SPLINE
SPL {X  -165.650, Y  +471.956, Z    +0.000, E1   -39.047, E3 +385632.686}
SPL {X  -165.650, Y  +478.019, Z    +0.000, E1   -39.139, E3 +385647.571}
SPL {X  -165.650, Y  +484.115, Z    +0.000, E1   -39.050, E3 +385663.332}
SPL {X  -165.650, Y  +488.489, Z    +0.000, E1   -39.102, E3 +385673.940}
SPL {X  -165.650, Y  +491.785, Z    +0.000, E1   -39.157, E3 +385681.913}
SPL {X  -165.650, Y  +496.519, Z    +0.000, E1   -39.062, E3 +385694.527}
SPL {X  -165.650, Y  +501.480, Z    +0.000, E1   -39.099, E3 +385706.684}
SPL {X  -165.650, Y  +505.989, Z    +0.000, E1   -39.067, E3 +385718.316}
SPL {X  -165.650, Y  +512.188, Z    +0.000, E1   -39.077, E3 +385733.959}
SPL {X  -165.650, Y  +516.634, Z    +0.000, E1   -39.035, E3 +385745.205}
SPL {X  -165.650, Y  +521.541, Z    +0.000, E1   -39.052, E3 +385757.752}
SPL {X  -165.650, Y  +527.474, Z    +0.000, E1   -39.169, E3 +385771.770}
SPL {X  -165.650, Y  +532.836, Z    +0.000, E1   -39.150, E3 +385785.552}
SPL {X  -165.650, Y  +537.667, Z    +0.000, E1   -38.986, E3 +385798.497}
SPL {X  -165.650, Y  +542.804, Z    +0.000, E1   -39.141, E3 +385810.681}
SPL {X  -165.650, Y  +547.280, Z    +0.000, E1   -38.965, E3 +385822.826}
SPL {X  -165.650, Y  +551.666, Z    +0.000, E1   -39.102, E3 +385833.144}
SPL {X  -165.650, Y  +557.612, Z    +0.000, E1   -39.166, E3 +385847.790}
SPL {X  -165.650, Y  +562.850, Z    +0.000, E1   -38.959, E3 +385862.149}
SPL {X  -165.650, Y  +568.257, Z    +0.000, E1   -39.077, E3 +385875.104}
SPL {X  -165.650, Y  +573.200, Z    +0.000, E1   -39.061, E3 +385887.639}
SPL {X  -165.650, Y  +578.240, Z    +0.000, E1   -39.117, E3 +385899.980}
SPL {X  -165.650, Y  +582.804, Z    +0.000, E1   -39.080, E3 +385911.687}
SPL {X  -165.650, Y  +587.640, Z    +0.000, E1   -39.069, E3 +385923.944}
SPL {X  -165.650, Y  +593.610, Z    +0.000, E1   -39.204, E3 +385938.217}
SPL {X  -165.650, Y  +599.021, Z    +0.000, E1   -38.950, E3 +385953.367}
SPL {X  -165.650, Y  +604.635, Z    +0.000, E1   -39.163, E3 +385966.144}
SPL {X  -165.650, Y  +608.365, Z    +0.000, E1   -39.063, E3 +385976.134}
SPL {X  -165.650, Y  +612.142, Z    +0.000, E1   -39.023, E3 +385985.864}
SPL {X  -165.650, Y  +616.635, Z    +0.000, E1   -39.260, E3 +385995.751}
SPL {X  -165.650, Y  +620.299, Z    +0.000, E1   -38.904, E3 +386007.138}
SPL {X  -165.650, Y  +625.662, Z    +0.000, E1   -39.189, E3 +386018.949}
SPL {X  -165.650, Y  +629.982, Z    +0.000, E1   -39.063, E3 +386030.550}
SPL {X  -165.650, Y  +635.019, Z    +0.000, E1   -39.106, E3 +386043.032}
SPL {X  -165.650, Y  +641.706, Z    +0.000, E1   -39.097, E3 +386060.099}
SPL {X  -165.650, Y  +648.294, Z    +0.000, E1   -39.142, E3 +386076.222}
SPL {X  -165.650, Y  +652.477, Z    +0.000, E1   -39.068, E3 +386087.124}
SPL {X  -165.650, Y  +656.920, Z    +0.000, E1   -39.120, E3 +386098.079}
SPL {X  -165.650, Y  +661.125, Z    +0.000, E1   -39.092, E3 +386108.728}
SPL {X  -165.650, Y  +664.437, Z    +0.000, E1   -39.114, E3 +386116.937}
SPL {X  -165.650, Y  +668.296, Z    +0.000, E1   -39.077, E3 +386126.909}
SPL {X  -165.650, Y  +673.138, Z    +0.000, E1   -39.196, E3 +386138.365}
SPL {X  -165.640, Y  +677.281, Z    +0.000, E1   -38.803, E3 +386151.254}
SPL {X  -165.389, Y  +684.794, Z    +0.000, E1   -39.261, E3 +386167.564}
SPL {X  -164.948, Y  +690.736, Z    +0.000, E1   -38.951, E3 +386184.233}
SPL {X  -164.363, Y  +696.109, Z    +0.000, E1   -38.853, E3 +386198.324}
SPL {X  -163.795, Y  +700.218, Z    +0.000, E1   -38.698, E3 +386209.531}
SPL {X  -162.937, Y  +705.358, Z    +0.000, E1   -38.703, E3 +386222.599}
SPL {X  -161.983, Y  +710.160, Z    +0.000, E1   -38.439, E3 +386236.093}
SPL {X  -161.163, Y  +713.794, Z    +0.000, E1   -38.390, E3 +386245.463}
SPL {X  -160.158, Y  +717.801, Z    +0.000, E1   -38.225, E3 +386256.593}
SPL {X  -155.870, Y  +731.575, Z    +0.000, E1   -42.661, E3 +386264.056}
SPL {X  -137.799, Y  +767.431, Z    +0.000, E1   -46.550, E3 +386320.566}
ENDSPLINE

SPLINE
SPL {X  -141.948, Y  +760.885, Z    +0.000, E1   -42.258, E3 +386352.702}
SPL {X  -160.264, Y  +717.397, Z    +0.000, E1   -24.835, E3 +386393.887}
SPL {X  -164.762, Y  +692.628, Z    +0.000, E1   -12.660, E3 +386397.139}
SPL {X  -165.581, Y  +680.274, Z    +0.000, E1    -5.699, E3 +386392.624}
SPL {X  -165.650, Y  +673.662, Z    +0.000, E1    -1.458, E3 +386389.583}
SPL {X  -165.650, Y  +670.254, Z    +0.000, E1    +1.045, E3 +386391.947}
SPL {X  -165.650, Y  +666.842, Z    +0.000, E1    +3.871, E3 +386390.049}
SPL {X  -165.650, Y  +661.513, Z    +0.000, E1    +8.695, E3 +386389.957}
SPL {X  -165.650, Y  +654.973, Z    +0.000, E1   +15.752, E3 +386387.363}
SPL {X  -165.650, Y  +648.120, Z    +0.000, E1   +22.794, E3 +386387.475}
SPL {X  -165.650, Y  +632.103, Z    +0.000, E1   +42.949, E3 +386374.433}
SPL {X  -165.650, Y  +609.948, Z    +0.000, E1   +49.636, E3 +386391.859}
SPL {X  -165.650, Y  +601.895, Z    +0.000, E1   +47.595, E3 +386409.529}
SPL {X  -165.650, Y  +568.828, Z    +0.000, E1   +48.639, E3 +386457.284}
ENDSPLINE

SPLINE
SPL {X  -165.650, Y  +587.144, Z    +0.000, E1   +39.840, E3 +386471.316}
ENDSPLINE

SPLINE
SPL {X  -165.650, Y  +582.480, Z    +0.000, E1   +38.929, E3 +386488.512}
SPL {X  -165.650, Y  +575.679, Z    +0.000, E1   +38.947, E3 +386505.587}
SPL {X  -165.650, Y  +569.616, Z    +0.000, E1   +38.966, E3 +386520.746}
SPL {X  -165.650, Y  +564.364, Z    +0.000, E1   +38.909, E3 +386534.398}
SPL {X  -165.650, Y  +559.065, Z    +0.000, E1   +38.883, E3 +386547.976}
SPL {X  -165.650, Y  +552.770, Z    +0.000, E1   +38.963, E3 +386563.537}
SPL {X  -165.650, Y  +546.277, Z    +0.000, E1   +38.910, E3 +386580.279}
SPL {X  -165.650, Y  +540.151, Z    +0.000, E1   +38.996, E3 +386595.208}
SPL {X  -165.650, Y  +534.008, Z    +0.000, E1   +38.962, E3 +386611.050}
SPL {X  -165.650, Y  +528.320, Z    +0.000, E1   +38.809, E3 +386626.287}
SPL {X  -165.650, Y  +522.377, Z    +0.000, E1   +38.974, E3 +386640.406}
ENDSPLINE

SPLINE
SPL {X  -165.650, Y  +539.854, Z    +0.000, E1   +28.090, E3 +386657.023}
ENDSPLINE

SPLINE
SPL {X  -165.650, Y  +534.443, Z    +0.000, E1   +28.969, E3 +386671.075}
SPL {X  -165.650, Y  +530.452, Z    +0.000, E1   +29.664, E3 +386680.808}
SPL {X  -165.650, Y  +525.298, Z    +0.000, E1   +30.602, E3 +386692.618}
SPL {X  -165.650, Y  +518.290, Z    +0.000, E1   +31.783, E3 +386708.511}
SPL {X  -165.650, Y  +512.706, Z    +0.000, E1   +32.573, E3 +386721.345}
SPL {X  -165.650, Y  +507.785, Z    +0.000, E1   +33.438, E3 +386731.282}
SPL {X  -165.650, Y  +501.257, Z    +0.000, E1   +34.478, E3 +386744.522}
SPL {X  -165.650, Y  +493.800, Z    +0.000, E1   +35.486, E3 +386760.010}
SPL {X  -165.650, Y  +485.583, Z    +0.000, E1   +36.670, E3 +386775.733}
SPL {X  -165.650, Y  +477.375, Z    +0.000, E1   +37.747, E3 +386791.252}
SPL {X  -165.650, Y  +469.901, Z    +0.000, E1   +38.767, E3 +386804.384}
SPL {X  -165.650, Y  +463.507, Z    +0.000, E1   +39.800, E3 +386814.131}
SPL {X  -165.650, Y  +460.803, Z    +0.000, E1   +39.417, E3 +386823.195}
SPL {X  -165.650, Y  +455.681, Z    +0.000, E1   +39.641, E3 +386834.516}
SPL {X  -165.650, Y  +451.332, Z    +0.000, E1   +39.738, E3 +386844.648}
SPL {X  -165.650, Y  +448.050, Z    +0.000, E1   +39.392, E3 +386854.814}
SPL {X  -165.650, Y  +442.946, Z    +0.000, E1   +39.866, E3 +386864.589}
SPL {X  -165.650, Y  +439.091, Z    +0.000, E1   +39.674, E3 +386875.207}
SPL {X  -165.650, Y  +434.131, Z    +0.000, E1   +39.643, E3 +386887.719}
SPL {X  -165.650, Y  +428.810, Z    +0.000, E1   +39.691, E3 +386900.482}
SPL {X  -165.650, Y  +424.197, Z    +0.000, E1   +39.695, E3 +386911.840}
SPL {X  -165.650, Y  +420.220, Z    +0.000, E1   +39.526, E3 +386922.635}
SPL {X  -165.650, Y  +414.177, Z    +0.000, E1   +39.693, E3 +386936.762}
SPL {X  -165.650, Y  +407.394, Z    +0.000, E1   +39.797, E3 +386952.717}
SPL {X  -165.650, Y  +402.798, Z    +0.000, E1   +39.651, E3 +386964.838}
SPL {X  -165.650, Y  +398.253, Z    +0.000, E1   +39.688, E3 +386975.842}
SPL {X  -165.650, Y  +393.720, Z    +0.000, E1   +39.686, E3 +386987.016}
SPL {X  -165.650, Y  +389.210, Z    +0.000, E1   +39.696, E3 +386998.066}
SPL {X  -165.650, Y  +384.878, Z    +0.000, E1   +39.631, E3 +387009.142}
SPL {X  -165.650, Y  +380.529, Z    +0.000, E1   +39.528, E3 +387020.529}
SPL {X  -165.618, Y  +375.240, Z    +0.000, E1   +39.617, E3 +387033.123}
SPL {X  -165.428, Y  +369.922, Z    +0.000, E1   +39.705, E3 +387045.664}
SPL {X  -165.216, Y  +366.519, Z    +0.000, E1   +39.498, E3 +387055.231}
SPL {X  -164.790, Y  +361.646, Z    +0.000, E1   +39.684, E3 +387066.226}
SPL {X  -164.317, Y  +357.530, Z    +0.000, E1   +39.402, E3 +387077.939}
SPL {X  -163.775, Y  +353.645, Z    +0.000, E1   +39.313, E3 +387088.110}
SPL {X  -163.109, Y  +349.595, Z    +0.000, E1   +39.290, E3 +387098.172}
SPL {X  -162.309, Y  +345.398, Z    +0.000, E1   +39.085, E3 +387109.835}
SPL {X  -161.467, Y  +341.510, Z    +0.000, E1   +38.980, E3 +387119.881}
SPL {X  -160.812, Y  +338.758, Z    +0.000, E1   +38.898, E3 +387127.138}
SPL {X  -159.926, Y  +335.332, Z    +0.000, E1   +38.809, E3 +387136.095}
SPL {X  -153.020, Y  +315.059, Z    +0.000, E1   +45.580, E3 +387142.827}
SPL {X  -148.632, Y  +305.368, Z    +0.000, E1   +40.700, E3 +387202.428}
SPL {X  -145.004, Y  +298.414, Z    +0.000, E1   +40.971, E3 +387227.164}
ENDSPLINE

SPLINE
SPL {X  -149.687, Y  +307.551, Z    +0.000, E1   +36.303, E3 +387262.596}
SPL {X  -158.807, Y  +331.381, Z    +0.000, E1   +26.928, E3 +387286.249}
SPL {X  -164.505, Y  +359.058, Z    +0.000, E1   +13.887, E3 +387275.010}
SPL {X  -165.494, Y  +371.321, Z    +0.000, E1    +7.176, E3 +387273.571}
SPL {X  -165.650, Y  +379.419, Z    +0.000, E1    +2.065, E3 +387271.252}
SPL {X  -165.650, Y  +383.176, Z    +0.000, E1    -0.610, E3 +387272.247}
SPL {X  -165.650, Y  +388.696, Z    +0.000, E1    -5.134, E3 +387270.524}
SPL {X  -165.650, Y  +394.663, Z    +0.000, E1   -10.843, E3 +387271.680}
SPL {X  -165.650, Y  +400.450, Z    +0.000, E1   -18.287, E3 +387262.979}
SPL {X  -165.650, Y  +409.248, Z    +0.000, E1   -26.478, E3 +387266.602}
SPL {X  -165.650, Y  +418.660, Z    +0.000, E1   -36.186, E3 +387264.078}
SPL {X  -165.650, Y  +444.260, Z    +0.000, E1   -47.328, E3 +387279.826}
SPL {X  -165.650, Y  +458.981, Z    +0.000, E1   -49.189, E3 +387295.369}
SPL {X  -165.650, Y  +493.049, Z    +0.000, E1   -51.657, E3 +387334.402}
ENDSPLINE

SPLINE
SPL {X  -165.650, Y  +468.984, Z    +0.000, E1   -41.461, E3 +387347.262}
SPL {X  -165.650, Y  +467.052, Z    +0.000, E1   -38.928, E3 +387357.877}
ENDSPLINE

SPLINE
SPL {X  -165.650, Y  +471.956, Z    +0.000, E1   -39.047, E3 +387369.528}
SPL {X  -165.650, Y  +478.019, Z    +0.000, E1   -39.139, E3 +387384.413}
SPL {X  -165.650, Y  +484.115, Z    +0.000, E1   -39.050, E3 +387400.174}
SPL {X  -165.650, Y  +490.374, Z    +0.000, E1   -39.169, E3 +387415.294}
SPL {X  -165.650, Y  +495.141, Z    +0.000, E1   -39.109, E3 +387427.450}
SPL {X  -165.650, Y  +497.824, Z    +0.000, E1   -38.944, E3 +387435.208}
SPL {X  -165.650, Y  +502.351, Z    +0.000, E1   -39.056, E3 +387446.092}
SPL {X  -165.650, Y  +508.180, Z    +0.000, E1   -39.157, E3 +387460.158}
SPL {X  -165.650, Y  +513.074, Z    +0.000, E1   -38.997, E3 +387473.375}
SPL {X  -165.650, Y  +518.439, Z    +0.000, E1   -39.071, E3 +387486.526}
SPL {X  -165.650, Y  +523.032, Z    +0.000, E1   -38.966, E3 +387498.662}
SPL {X  -165.650, Y  +528.401, Z    +0.000, E1   -39.135, E3 +387511.262}
SPL {X  -165.650, Y  +533.857, Z    +0.000, E1   -39.163, E3 +387524.768}
SPL {X  -165.650, Y  +539.651, Z    +0.000, E1   -39.087, E3 +387539.912}
SPL {X  -165.650, Y  +544.603, Z    +0.000, E1   -39.103, E3 +387552.088}
SPL {X  -165.650, Y  +547.280, Z    +0.000, E1   -38.965, E3 +387559.668}
SPL {X  -165.650, Y  +551.666, Z    +0.000, E1   -39.102, E3 +387569.986}
SPL {X  -165.650, Y  +555.880, Z    +0.000, E1   -39.094, E3 +387580.557}
SPL {X  -165.650, Y  +559.255, Z    +0.000, E1   -39.167, E3 +387588.593}
SPL {X  -165.650, Y  +562.850, Z    +0.000, E1   -38.959, E3 +387598.991}
SPL {X  -165.650, Y  +568.257, Z    +0.000, E1   -39.077, E3 +387611.946}
SPL {X  -165.650, Y  +573.200, Z    +0.000, E1   -39.061, E3 +387624.481}
SPL {X  -165.650, Y  +578.240, Z    +0.000, E1   -39.117, E3 +387636.822}
SPL {X  -165.650, Y  +582.804, Z    +0.000, E1   -39.080, E3 +387648.529}
SPL {X  -165.650, Y  +587.640, Z    +0.000, E1   -39.069, E3 +387660.786}
SPL {X  -165.650, Y  +593.610, Z    +0.000, E1   -39.204, E3 +387675.060}
SPL {X  -165.650, Y  +599.021, Z    +0.000, E1   -38.950, E3 +387690.209}
SPL {X  -165.650, Y  +604.635, Z    +0.000, E1   -39.163, E3 +387702.986}
SPL {X  -165.650, Y  +608.365, Z    +0.000, E1   -39.063, E3 +387712.976}
SPL {X  -165.650, Y  +612.142, Z    +0.000, E1   -39.023, E3 +387722.706}
SPL {X  -165.650, Y  +616.635, Z    +0.000, E1   -39.260, E3 +387732.593}
SPL {X  -165.650, Y  +620.299, Z    +0.000, E1   -38.904, E3 +387743.980}
SPL {X  -165.650, Y  +625.662, Z    +0.000, E1   -39.189, E3 +387755.791}
SPL {X  -165.650, Y  +629.982, Z    +0.000, E1   -39.063, E3 +387767.392}
SPL {X  -165.650, Y  +635.019, Z    +0.000, E1   -39.106, E3 +387779.874}
SPL {X  -165.650, Y  +640.403, Z    +0.000, E1   -39.127, E3 +387793.270}
SPL {X  -165.650, Y  +645.443, Z    +0.000, E1   -39.032, E3 +387806.575}
SPL {X  -165.650, Y  +651.452, Z    +0.000, E1   -39.128, E3 +387821.144}
SPL {X  -165.650, Y  +656.920, Z    +0.000, E1   -39.120, E3 +387834.921}
SPL {X  -165.650, Y  +661.125, Z    +0.000, E1   -39.092, E3 +387845.570}
SPL {X  -165.650, Y  +664.437, Z    +0.000, E1   -39.114, E3 +387853.779}
SPL {X  -165.650, Y  +668.296, Z    +0.000, E1   -39.077, E3 +387863.751}
SPL {X  -165.650, Y  +673.138, Z    +0.000, E1   -39.196, E3 +387875.207}
SPL {X  -165.640, Y  +677.281, Z    +0.000, E1   -38.803, E3 +387888.096}
SPL {X  -165.461, Y  +683.414, Z    +0.000, E1   -39.212, E3 +387901.080}
SPL {X  -165.241, Y  +687.126, Z    +0.000, E1   -39.221, E3 +387910.223}
SPL {X  -164.948, Y  +690.736, Z    +0.000, E1   -38.951, E3 +387921.075}
SPL {X  -164.363, Y  +696.109, Z    +0.000, E1   -38.853, E3 +387935.166}
SPL {X  -163.795, Y  +700.218, Z    +0.000, E1   -38.698, E3 +387946.373}
SPL {X  -162.937, Y  +705.358, Z    +0.000, E1   -38.703, E3 +387959.441}
SPL {X  -161.983, Y  +710.160, Z    +0.000, E1   -38.439, E3 +387972.935}
SPL {X  -160.874, Y  +714.989, Z    +0.000, E1   -38.205, E3 +387986.596}
SPL {X  -159.557, Y  +720.012, Z    +0.000, E1   -38.534, E3 +387997.137}
SPL {X  -155.870, Y  +731.575, Z    +0.000, E1   -42.661, E3 +388000.898}
SPL {X  -137.799, Y  +767.431, Z    +0.000, E1   -46.550, E3 +388057.408}
ENDSPLINE

SPLINE
SPL {X  -141.948, Y  +760.885, Z    +0.000, E1   -42.258, E3 +388089.544}
SPL {X  -160.264, Y  +717.397, Z    +0.000, E1   -24.835, E3 +388130.729}
SPL {X  -164.457, Y  +695.345, Z    +0.000, E1   -14.031, E3 +388137.670}
SPL {X  -165.312, Y  +686.072, Z    +0.000, E1    -9.096, E3 +388130.764}
SPL {X  -165.625, Y  +678.398, Z    +0.000, E1    -4.508, E3 +388128.506}
SPL {X  -165.650, Y  +673.662, Z    +0.000, E1    -1.458, E3 +388126.425}
SPL {X  -165.650, Y  +670.254, Z    +0.000, E1    +1.045, E3 +388128.789}
SPL {X  -165.650, Y  +666.842, Z    +0.000, E1    +3.871, E3 +388126.891}
SPL {X  -165.650, Y  +662.773, Z    +0.000, E1    +7.549, E3 +388127.036}
SPL {X  -165.650, Y  +656.581, Z    +0.000, E1   +13.870, E3 +388125.086}
SPL {X  -165.650, Y  +648.120, Z    +0.000, E1   +22.794, E3 +388124.317}
SPL {X  -165.650, Y  +632.103, Z    +0.000, E1   +42.949, E3 +388111.275}
SPL {X  -165.650, Y  +609.948, Z    +0.000, E1   +49.636, E3 +388128.701}
SPL {X  -165.650, Y  +601.895, Z    +0.000, E1   +47.595, E3 +388146.371}
SPL {X  -165.650, Y  +568.828, Z    +0.000, E1   +48.639, E3 +388194.126}
ENDSPLINE

SPLINE
SPL {X  -165.650, Y  +587.144, Z    +0.000, E1   +39.840, E3 +388208.158}
ENDSPLINE

SPLINE
SPL {X  -165.650, Y  +582.480, Z    +0.000, E1   +38.929, E3 +388225.354}
SPL {X  -165.650, Y  +576.923, Z    +0.000, E1   +38.908, E3 +388239.384}
SPL {X  -165.650, Y  +570.800, Z    +0.000, E1   +39.001, E3 +388254.559}
SPL {X  -165.650, Y  +564.364, Z    +0.000, E1   +38.909, E3 +388271.241}
SPL {X  -165.650, Y  +559.065, Z    +0.000, E1   +38.883, E3 +388284.819}
SPL {X  -165.650, Y  +554.358, Z    +0.000, E1   +38.887, E3 +388296.660}
SPL {X  -165.650, Y  +549.409, Z    +0.000, E1   +38.884, E3 +388309.341}
SPL {X  -165.650, Y  +542.772, Z    +0.000, E1   +39.054, E3 +388325.137}
SPL {X  -165.650, Y  +537.647, Z    +0.000, E1   +38.838, E3 +388339.299}
SPL {X  -165.650, Y  +532.636, Z    +0.000, E1   +39.009, E3 +388350.945}
SPL {X  -165.650, Y  +528.320, Z    +0.000, E1   +38.809, E3 +388363.129}
SPL {X  -165.650, Y  +522.377, Z    +0.000, E1   +38.974, E3 +388377.249}
ENDSPLINE

SPLINE
SPL {X  -165.650, Y  +541.168, Z    +0.000, E1   +27.957, E3 +388389.588}
ENDSPLINE

SPLINE
SPL {X  -165.650, Y  +536.052, Z    +0.000, E1   +28.653, E3 +388404.223}
SPL {X  -165.650, Y  +530.452, Z    +0.000, E1   +29.664, E3 +388417.650}
SPL {X  -165.650, Y  +523.712, Z    +0.000, E1   +30.911, E3 +388432.932}
SPL {X  -165.650, Y  +516.975, Z    +0.000, E1   +31.942, E3 +388448.526}
SPL {X  -165.650, Y  +512.706, Z    +0.000, E1   +32.573, E3 +388458.187}
SPL {X  -165.650, Y  +507.785, Z    +0.000, E1   +33.438, E3 +388468.124}
SPL {X  -165.650, Y  +501.257, Z    +0.000, E1   +34.478, E3 +388481.364}
SPL {X  -165.650, Y  +495.236, Z    +0.000, E1   +35.288, E3 +388493.870}
SPL {X  -165.650, Y  +488.684, Z    +0.000, E1   +36.217, E3 +388506.766}
SPL {X  -165.650, Y  +481.130, Z    +0.000, E1   +37.251, E3 +388521.075}
SPL {X  -165.650, Y  +475.455, Z    +0.000, E1   +37.964, E3 +388531.732}
SPL {X  -165.650, Y  +469.901, Z    +0.000, E1   +38.767, E3 +388541.226}
SPL {X  -165.650, Y  +465.276, Z    +0.000, E1   +39.067, E3 +388551.103}
SPL {X  -165.650, Y  +459.623, Z    +0.000, E1   +39.919, E3 +388560.038}
SPL {X  -165.650, Y  +455.681, Z    +0.000, E1   +39.641, E3 +388571.358}
SPL {X  -165.650, Y  +451.332, Z    +0.000, E1   +39.738, E3 +388581.491}
SPL {X  -165.650, Y  +448.050, Z    +0.000, E1   +39.392, E3 +388591.656}
SPL {X  -165.650, Y  +442.946, Z    +0.000, E1   +39.866, E3 +388601.431}
SPL {X  -165.650, Y  +439.091, Z    +0.000, E1   +39.674, E3 +388612.049}
SPL {X  -165.650, Y  +435.404, Z    +0.000, E1   +39.549, E3 +388621.886}
SPL {X  -165.650, Y  +429.757, Z    +0.000, E1   +39.737, E3 +388634.835}
SPL {X  -165.650, Y  +424.197, Z    +0.000, E1   +39.695, E3 +388648.682}
SPL {X  -165.650, Y  +420.220, Z    +0.000, E1   +39.526, E3 +388659.477}
SPL {X  -165.650, Y  +415.675, Z    +0.000, E1   +39.706, E3 +388669.639}
SPL {X  -165.650, Y  +412.313, Z    +0.000, E1   +39.567, E3 +388678.717}
SPL {X  -165.650, Y  +407.394, Z    +0.000, E1   +39.797, E3 +388689.559}
SPL {X  -165.650, Y  +402.798, Z    +0.000, E1   +39.651, E3 +388701.681}
SPL {X  -165.650, Y  +398.253, Z    +0.000, E1   +39.688, E3 +388712.684}
SPL {X  -165.650, Y  +393.720, Z    +0.000, E1   +39.686, E3 +388723.858}
SPL {X  -165.650, Y  +389.210, Z    +0.000, E1   +39.696, E3 +388734.908}
SPL {X  -165.650, Y  +384.878, Z    +0.000, E1   +39.631, E3 +388745.985}
SPL {X  -165.650, Y  +380.529, Z    +0.000, E1   +39.528, E3 +388757.371}
SPL {X  -165.618, Y  +375.240, Z    +0.000, E1   +39.617, E3 +388769.965}
SPL {X  -165.428, Y  +369.922, Z    +0.000, E1   +39.705, E3 +388782.507}
SPL {X  -165.216, Y  +366.519, Z    +0.000, E1   +39.498, E3 +388792.073}
SPL {X  -164.790, Y  +361.646, Z    +0.000, E1   +39.684, E3 +388803.068}
SPL {X  -164.317, Y  +357.530, Z    +0.000, E1   +39.402, E3 +388814.781}
SPL {X  -163.775, Y  +353.645, Z    +0.000, E1   +39.313, E3 +388824.952}
SPL {X  -162.932, Y  +348.615, Z    +0.000, E1   +39.259, E3 +388837.716}
SPL {X  -162.143, Y  +344.596, Z    +0.000, E1   +39.019, E3 +388848.933}
SPL {X  -161.093, Y  +339.912, Z    +0.000, E1   +38.966, E3 +388860.884}
SPL {X  -159.926, Y  +335.332, Z    +0.000, E1   +38.809, E3 +388872.937}
SPL {X  -153.020, Y  +315.059, Z    +0.000, E1   +45.580, E3 +388879.669}
SPL {X  -148.632, Y  +305.368, Z    +0.000, E1   +40.700, E3 +388939.271}
SPL {X  -145.004, Y  +298.414, Z    +0.000, E1   +40.971, E3 +388964.006}
ENDSPLINE

SPLINE
SPL {X  -149.687, Y  +307.551, Z    +0.000, E1   +36.303, E3 +388999.438}
SPL {X  -158.807, Y  +331.381, Z    +0.000, E1   +26.928, E3 +389023.091}
SPL {X  -164.505, Y  +359.058, Z    +0.000, E1   +13.887, E3 +389011.853}
SPL {X  -165.494, Y  +371.321, Z    +0.000, E1    +7.176, E3 +389010.413}
SPL {X  -165.650, Y  +379.419, Z    +0.000, E1    +2.065, E3 +389008.094}
SPL {X  -165.650, Y  +383.176, Z    +0.000, E1    -0.610, E3 +389009.090}
SPL {X  -165.650, Y  +388.696, Z    +0.000, E1    -5.134, E3 +389007.366}
SPL {X  -165.650, Y  +394.663, Z    +0.000, E1   -10.843, E3 +389008.522}
SPL {X  -165.650, Y  +400.450, Z    +0.000, E1   -18.287, E3 +388999.821}
SPL {X  -165.650, Y  +409.248, Z    +0.000, E1   -26.478, E3 +389003.444}
SPL {X  -165.650, Y  +418.660, Z    +0.000, E1   -36.186, E3 +389000.920}
SPL {X  -165.650, Y  +444.260, Z    +0.000, E1   -47.328, E3 +389016.668}
SPL {X  -165.650, Y  +458.981, Z    +0.000, E1   -49.189, E3 +389032.212}
SPL {X  -165.650, Y  +493.049, Z    +0.000, E1   -51.657, E3 +389071.244}
ENDSPLINE

SPLINE
SPL {X  -165.650, Y  +468.984, Z    +0.000, E1   -41.461, E3 +389084.105}
SPL {X  -165.650, Y  +467.052, Z    +0.000, E1   -38.928, E3 +389094.719}
ENDSPLINE

SPLINE
SPL {X  -165.650, Y  +471.956, Z    +0.000, E1   -39.047, E3 +389106.370}
SPL {X  -165.650, Y  +478.019, Z    +0.000, E1   -39.139, E3 +389121.255}
SPL {X  -165.650, Y  +484.115, Z    +0.000, E1   -39.050, E3 +389137.016}
SPL {X  -165.650, Y  +490.374, Z    +0.000, E1   -39.169, E3 +389152.136}
SPL {X  -165.650, Y  +495.141, Z    +0.000, E1   -39.109, E3 +389164.292}
SPL {X  -165.650, Y  +499.941, Z    +0.000, E1   -39.068, E3 +389176.821}
SPL {X  -165.650, Y  +505.989, Z    +0.000, E1   -39.067, E3 +389192.001}
SPL {X  -165.650, Y  +512.188, Z    +0.000, E1   -39.077, E3 +389207.643}
SPL {X  -165.650, Y  +518.439, Z    +0.000, E1   -39.071, E3 +389223.368}
SPL {X  -165.650, Y  +523.032, Z    +0.000, E1   -38.966, E3 +389235.504}
SPL {X  -165.650, Y  +528.401, Z    +0.000, E1   -39.135, E3 +389248.104}
SPL {X  -165.650, Y  +533.857, Z    +0.000, E1   -39.163, E3 +389261.610}
SPL {X  -165.650, Y  +539.651, Z    +0.000, E1   -39.087, E3 +389276.754}
SPL {X  -165.650, Y  +546.018, Z    +0.000, E1   -39.065, E3 +389292.879}
SPL {X  -165.650, Y  +551.666, Z    +0.000, E1   -39.102, E3 +389306.828}
SPL {X  -165.650, Y  +557.612, Z    +0.000, E1   -39.166, E3 +389321.474}
SPL {X  -165.650, Y  +562.850, Z    +0.000, E1   -38.959, E3 +389335.833}
SPL {X  -165.650, Y  +568.257, Z    +0.000, E1   -39.077, E3 +389348.788}
SPL {X  -165.650, Y  +573.200, Z    +0.000, E1   -39.061, E3 +389361.323}
SPL {X  -165.650, Y  +578.240, Z    +0.000, E1   -39.117, E3 +389373.664}
SPL {X  -165.650, Y  +582.804, Z    +0.000, E1   -39.080, E3 +389385.371}
SPL {X  -165.650, Y  +587.640, Z    +0.000, E1   -39.069, E3 +389397.628}
SPL {X  -165.650, Y  +593.610, Z    +0.000, E1   -39.204, E3 +389411.902}
SPL {X  -165.650, Y  +599.021, Z    +0.000, E1   -38.950, E3 +389427.051}
SPL {X  -165.650, Y  +604.635, Z    +0.000, E1   -39.163, E3 +389439.828}
SPL {X  -165.650, Y  +608.365, Z    +0.000, E1   -39.063, E3 +389449.818}
SPL {X  -165.650, Y  +613.618, Z    +0.000, E1   -39.137, E3 +389462.682}
SPL {X  -165.650, Y  +619.584, Z    +0.000, E1   -39.045, E3 +389478.319}
SPL {X  -165.650, Y  +625.662, Z    +0.000, E1   -39.189, E3 +389492.633}
SPL {X  -165.650, Y  +629.982, Z    +0.000, E1   -39.063, E3 +389504.234}
SPL {X  -165.650, Y  +635.019, Z    +0.000, E1   -39.106, E3 +389516.716}
SPL {X  -165.650, Y  +641.706, Z    +0.000, E1   -39.097, E3 +389533.783}
SPL {X  -165.650, Y  +648.294, Z    +0.000, E1   -39.142, E3 +389549.906}
SPL {X  -165.650, Y  +652.477, Z    +0.000, E1   -39.068, E3 +389560.808}
SPL {X  -165.650, Y  +656.920, Z    +0.000, E1   -39.120, E3 +389571.763}
SPL {X  -165.650, Y  +661.125, Z    +0.000, E1   -39.092, E3 +389582.412}
SPL {X  -165.650, Y  +664.437, Z    +0.000, E1   -39.114, E3 +389590.621}
SPL {X  -165.650, Y  +668.296, Z    +0.000, E1   -39.077, E3 +389600.593}
SPL {X  -165.650, Y  +673.138, Z    +0.000, E1   -39.196, E3 +389612.049}
SPL {X  -165.640, Y  +677.281, Z    +0.000, E1   -38.803, E3 +389624.938}
SPL {X  -165.461, Y  +683.414, Z    +0.000, E1   -39.212, E3 +389637.922}
SPL {X  -165.139, Y  +688.497, Z    +0.000, E1   -39.013, E3 +389651.974}
SPL {X  -164.582, Y  +694.282, Z    +0.000, E1   -38.975, E3 +389666.722}
SPL {X  -163.926, Y  +699.336, Z    +0.000, E1   -38.767, E3 +389680.700}
SPL {X  -162.937, Y  +705.358, Z    +0.000, E1   -38.703, E3 +389696.283}
SPL {X  -161.983, Y  +710.160, Z    +0.000, E1   -38.439, E3 +389709.777}
SPL {X  -161.163, Y  +713.794, Z    +0.000, E1   -38.390, E3 +389719.147}
SPL {X  -160.158, Y  +717.801, Z    +0.000, E1   -38.225, E3 +389730.277}
SPL {X  -155.870, Y  +731.575, Z    +0.000, E1   -42.661, E3 +389737.740}
SPL {X  -137.799, Y  +767.431, Z    +0.000, E1   -46.550, E3 +389794.250}
ENDSPLINE

SPLINE
SPL {X  -141.948, Y  +760.885, Z    +0.000, E1   -42.258, E3 +389826.386}
SPL {X  -160.264, Y  +717.397, Z    +0.000, E1   -24.835, E3 +389867.571}
SPL {X  -164.762, Y  +692.628, Z    +0.000, E1   -12.660, E3 +389870.824}
SPL {X  -165.581, Y  +680.274, Z    +0.000, E1    -5.699, E3 +389866.308}
SPL {X  -165.650, Y  +673.662, Z    +0.000, E1    -1.458, E3 +389863.267}
SPL {X  -165.650, Y  +670.254, Z    +0.000, E1    +1.045, E3 +389865.631}
SPL {X  -165.650, Y  +666.842, Z    +0.000, E1    +3.871, E3 +389863.733}
SPL {X  -165.650, Y  +661.513, Z    +0.000, E1    +8.695, E3 +389863.641}
SPL {X  -165.650, Y  +654.973, Z    +0.000, E1   +15.752, E3 +389861.048}
SPL {X  -165.650, Y  +648.120, Z    +0.000, E1   +22.794, E3 +389861.159}
SPL {X  -165.650, Y  +632.103, Z    +0.000, E1   +42.949, E3 +389848.117}
SPL {X  -165.650, Y  +609.948, Z    +0.000, E1   +49.636, E3 +389865.543}
SPL {X  -165.650, Y  +601.895, Z    +0.000, E1   +47.595, E3 +389883.213}
SPL {X  -165.650, Y  +568.828, Z    +0.000, E1   +48.639, E3 +389930.968}
ENDSPLINE

SPLINE
SPL {X  -165.650, Y  +587.144, Z    +0.000, E1   +39.840, E3 +389945.000}
ENDSPLINE

SPLINE
SPL {X  -165.650, Y  +582.480, Z    +0.000, E1   +38.929, E3 +389962.196}
SPL {X  -165.650, Y  +575.679, Z    +0.000, E1   +38.947, E3 +389979.272}
SPL {X  -165.650, Y  +569.616, Z    +0.000, E1   +38.966, E3 +389994.430}
SPL {X  -165.650, Y  +564.364, Z    +0.000, E1   +38.909, E3 +390008.083}
SPL {X  -165.650, Y  +559.065, Z    +0.000, E1   +38.883, E3 +390021.661}
SPL {X  -165.650, Y  +552.770, Z    +0.000, E1   +38.963, E3 +390037.221}
SPL {X  -165.650, Y  +546.277, Z    +0.000, E1   +38.910, E3 +390053.963}
SPL {X  -165.650, Y  +540.151, Z    +0.000, E1   +38.996, E3 +390068.893}
SPL {X  -165.650, Y  +534.008, Z    +0.000, E1   +38.962, E3 +390084.735}
SPL {X  -165.650, Y  +528.320, Z    +0.000, E1   +38.809, E3 +390099.971}
SPL {X  -165.650, Y  +522.377, Z    +0.000, E1   +38.974, E3 +390114.091}
ENDSPLINE

SPLINE
SPL {X  -165.650, Y  +539.854, Z    +0.000, E1   +28.090, E3 +390130.708}
ENDSPLINE

SPLINE
SPL {X  -165.650, Y  +534.443, Z    +0.000, E1   +28.969, E3 +390144.759}
SPL {X  -165.650, Y  +530.452, Z    +0.000, E1   +29.664, E3 +390154.492}
SPL {X  -165.650, Y  +525.298, Z    +0.000, E1   +30.602, E3 +390166.303}
SPL {X  -165.650, Y  +518.290, Z    +0.000, E1   +31.783, E3 +390182.195}
SPL {X  -165.650, Y  +512.706, Z    +0.000, E1   +32.573, E3 +390195.029}
SPL {X  -165.650, Y  +507.785, Z    +0.000, E1   +33.438, E3 +390204.967}
SPL {X  -165.650, Y  +501.257, Z    +0.000, E1   +34.478, E3 +390218.206}
SPL {X  -165.650, Y  +493.800, Z    +0.000, E1   +35.486, E3 +390233.694}
SPL {X  -165.650, Y  +485.583, Z    +0.000, E1   +36.670, E3 +390249.417}
SPL {X  -165.650, Y  +477.375, Z    +0.000, E1   +37.747, E3 +390264.936}
SPL {X  -165.650, Y  +469.901, Z    +0.000, E1   +38.767, E3 +390278.068}
SPL {X  -165.650, Y  +463.507, Z    +0.000, E1   +39.800, E3 +390287.816}
SPL {X  -165.650, Y  +460.803, Z    +0.000, E1   +39.417, E3 +390296.879}
SPL {X  -165.650, Y  +455.681, Z    +0.000, E1   +39.641, E3 +390308.200}
SPL {X  -165.650, Y  +451.332, Z    +0.000, E1   +39.738, E3 +390318.333}
SPL {X  -165.650, Y  +448.050, Z    +0.000, E1   +39.392, E3 +390328.498}
SPL {X  -165.650, Y  +442.946, Z    +0.000, E1   +39.866, E3 +390338.273}
SPL {X  -165.650, Y  +439.091, Z    +0.000, E1   +39.674, E3 +390348.891}
SPL {X  -165.650, Y  +434.131, Z    +0.000, E1   +39.643, E3 +390361.404}
SPL {X  -165.650, Y  +428.810, Z    +0.000, E1   +39.691, E3 +390374.166}
SPL {X  -165.650, Y  +424.197, Z    +0.000, E1   +39.695, E3 +390385.524}
SPL {X  -165.650, Y  +420.220, Z    +0.000, E1   +39.526, E3 +390396.320}
SPL {X  -165.650, Y  +414.177, Z    +0.000, E1   +39.693, E3 +390410.446}
SPL {X  -165.650, Y  +407.394, Z    +0.000, E1   +39.797, E3 +390426.401}
SPL {X  -165.650, Y  +402.798, Z    +0.000, E1   +39.651, E3 +390438.523}
SPL {X  -165.650, Y  +398.253, Z    +0.000, E1   +39.688, E3 +390449.526}
SPL {X  -165.650, Y  +393.720, Z    +0.000, E1   +39.686, E3 +390460.701}
SPL {X  -165.650, Y  +389.210, Z    +0.000, E1   +39.696, E3 +390471.750}
SPL {X  -165.650, Y  +384.878, Z    +0.000, E1   +39.631, E3 +390482.827}
SPL {X  -165.650, Y  +380.529, Z    +0.000, E1   +39.528, E3 +390494.213}
SPL {X  -165.618, Y  +375.240, Z    +0.000, E1   +39.617, E3 +390506.807}
SPL {X  -165.428, Y  +369.922, Z    +0.000, E1   +39.705, E3 +390519.349}
SPL {X  -165.216, Y  +366.519, Z    +0.000, E1   +39.498, E3 +390528.916}
SPL {X  -164.790, Y  +361.646, Z    +0.000, E1   +39.684, E3 +390539.910}
SPL {X  -164.317, Y  +357.530, Z    +0.000, E1   +39.402, E3 +390551.623}
SPL {X  -163.775, Y  +353.645, Z    +0.000, E1   +39.313, E3 +390561.794}
SPL {X  -163.109, Y  +349.595, Z    +0.000, E1   +39.290, E3 +390571.856}
SPL {X  -162.309, Y  +345.398, Z    +0.000, E1   +39.085, E3 +390583.520}
SPL {X  -161.467, Y  +341.510, Z    +0.000, E1   +38.980, E3 +390593.565}
SPL {X  -160.812, Y  +338.758, Z    +0.000, E1   +38.898, E3 +390600.822}
SPL {X  -159.926, Y  +335.332, Z    +0.000, E1   +38.809, E3 +390609.780}
SPL {X  -153.020, Y  +315.059, Z    +0.000, E1   +45.580, E3 +390616.511}
SPL {X  -148.632, Y  +305.368, Z    +0.000, E1   +40.700, E3 +390676.113}
SPL {X  -145.004, Y  +298.414, Z    +0.000, E1   +40.971, E3 +390700.848}
ENDSPLINE

SPLINE
SPL {X  -149.687, Y  +307.551, Z    +0.000, E1   +36.303, E3 +390736.280}
SPL {X  -158.807, Y  +331.381, Z    +0.000, E1   +26.928, E3 +390759.933}
SPL {X  -164.505, Y  +359.058, Z    +0.000, E1   +13.887, E3 +390748.695}
SPL {X  -165.334, Y  +368.271, Z    +0.000, E1    +8.886, E3 +390746.533}
SPL {X  -165.596, Y  +374.277, Z    +0.000, E1    +5.306, E3 +390747.915}
SPL {X  -165.650, Y  +379.419, Z    +0.000, E1    +2.065, E3 +390744.937}
SPL {X  -165.650, Y  +383.176, Z    +0.000, E1    -0.610, E3 +390745.932}
SPL {X  -165.650, Y  +387.435, Z    +0.000, E1    -4.104, E3 +390744.292}
SPL {X  -165.650, Y  +393.422, Z    +0.000, E1    -9.605, E3 +390744.849}
SPL {X  -165.650, Y  +400.450, Z    +0.000, E1   -18.287, E3 +390736.663}
SPL {X  -165.650, Y  +409.248, Z    +0.000, E1   -26.478, E3 +390740.286}
SPL {X  -165.650, Y  +418.660, Z    +0.000, E1   -36.186, E3 +390737.762}
SPL {X  -165.650, Y  +444.260, Z    +0.000, E1   -47.328, E3 +390753.510}
SPL {X  -165.650, Y  +458.981, Z    +0.000, E1   -49.189, E3 +390769.054}
SPL {X  -165.650, Y  +493.049, Z    +0.000, E1   -51.657, E3 +390808.087}
ENDSPLINE

SPLINE
SPL {X  -165.650, Y  +468.984, Z    +0.000, E1   -41.461, E3 +390820.947}
SPL {X  -165.650, Y  +467.052, Z    +0.000, E1   -38.928, E3 +390831.562}
ENDSPLINE

SPLINE
SPL {X  -165.650, Y  +471.956, Z    +0.000, E1   -39.047, E3 +390843.213}
SPL {X  -165.650, Y  +476.270, Z    +0.000, E1   -39.142, E3 +390853.469}
SPL {X  -165.650, Y  +480.876, Z    +0.000, E1   -39.050, E3 +390865.751}
SPL {X  -165.650, Y  +487.054, Z    +0.000, E1   -39.118, E3 +390880.890}
SPL {X  -165.650, Y  +491.785, Z    +0.000, E1   -39.157, E3 +390892.439}
SPL {X  -165.650, Y  +496.519, Z    +0.000, E1   -39.062, E3 +390905.053}
SPL {X  -165.650, Y  +501.480, Z    +0.000, E1   -39.099, E3 +390917.210}
SPL {X  -165.650, Y  +505.989, Z    +0.000, E1   -39.067, E3 +390928.843}
SPL {X  -165.650, Y  +512.188, Z    +0.000, E1   -39.077, E3 +390944.485}
SPL {X  -165.650, Y  +516.634, Z    +0.000, E1   -39.035, E3 +390955.731}
SPL {X  -165.650, Y  +521.541, Z    +0.000, E1   -39.052, E3 +390968.278}
SPL {X  -165.650, Y  +527.474, Z    +0.000, E1   -39.169, E3 +390982.296}
SPL {X  -165.650, Y  +532.836, Z    +0.000, E1   -39.150, E3 +390996.078}
SPL {X  -165.650, Y  +537.667, Z    +0.000, E1   -38.986, E3 +391009.023}
SPL {X  -165.650, Y  +541.183, Z    +0.000, E1   -39.101, E3 +391017.210}
SPL {X  -165.650, Y  +546.018, Z    +0.000, E1   -39.065, E3 +391029.721}
SPL {X  -165.650, Y  +551.666, Z    +0.000, E1   -39.102, E3 +391043.670}
SPL {X  -165.650, Y  +557.612, Z    +0.000, E1   -39.166, E3 +391058.317}
SPL {X  -165.650, Y  +562.850, Z    +0.000, E1   -38.959, E3 +391072.675}
SPL {X  -165.650, Y  +568.257, Z    +0.000, E1   -39.077, E3 +391085.630}
SPL {X  -165.650, Y  +573.200, Z    +0.000, E1   -39.061, E3 +391098.165}
SPL {X  -165.650, Y  +578.240, Z    +0.000, E1   -39.117, E3 +391110.506}
SPL {X  -165.650, Y  +582.804, Z    +0.000, E1   -39.080, E3 +391122.213}
SPL {X  -165.650, Y  +587.640, Z    +0.000, E1   -39.069, E3 +391134.470}
SPL {X  -165.650, Y  +593.610, Z    +0.000, E1   -39.204, E3 +391148.744}
SPL {X  -165.650, Y  +599.021, Z    +0.000, E1   -38.950, E3 +391163.893}
SPL {X  -165.650, Y  +604.635, Z    +0.000, E1   -39.163, E3 +391176.670}
SPL {X  -165.650, Y  +608.365, Z    +0.000, E1   -39.063, E3 +391186.660}
SPL {X  -165.650, Y  +612.142, Z    +0.000, E1   -39.023, E3 +391196.390}
SPL {X  -165.650, Y  +616.635, Z    +0.000, E1   -39.260, E3 +391206.278}
SPL {X  -165.650, Y  +620.299, Z    +0.000, E1   -38.904, E3 +391217.664}
SPL {X  -165.650, Y  +625.662, Z    +0.000, E1   -39.189, E3 +391229.475}
SPL {X  -165.650, Y  +629.982, Z    +0.000, E1   -39.063, E3 +391241.077}
SPL {X  -165.650, Y  +634.317, Z    +0.000, E1   -39.239, E3 +391250.867}
SPL {X  -165.650, Y  +639.215, Z    +0.000, E1   -39.074, E3 +391264.392}
SPL {X  -165.650, Y  +643.707, Z    +0.000, E1   -38.911, E3 +391276.492}
SPL {X  -165.650, Y  +648.294, Z    +0.000, E1   -39.142, E3 +391286.748}
SPL {X  -165.650, Y  +652.477, Z    +0.000, E1   -39.068, E3 +391297.650}
SPL {X  -165.650, Y  +656.920, Z    +0.000, E1   -39.120, E3 +391308.606}
SPL {X  -165.650, Y  +662.945, Z    +0.000, E1   -39.141, E3 +391323.711}
SPL {X  -165.650, Y  +668.296, Z    +0.000, E1   -39.077, E3 +391337.436}
SPL {X  -165.650, Y  +673.138, Z    +0.000, E1   -39.196, E3 +391348.891}
SPL {X  -165.640, Y  +677.281, Z    +0.000, E1   -38.803, E3 +391361.780}
SPL {X  -165.461, Y  +683.414, Z    +0.000, E1   -39.212, E3 +391374.764}
SPL {X  -165.139, Y  +688.497, Z    +0.000, E1   -39.013, E3 +391388.816}
SPL {X  -164.582, Y  +694.282, Z    +0.000, E1   -38.975, E3 +391403.564}
SPL {X  -163.926, Y  +699.336, Z    +0.000, E1   -38.767, E3 +391417.542}
SPL {X  -163.214, Y  +703.806, Z    +0.000, E1   -38.755, E3 +391428.727}
SPL {X  -162.700, Y  +706.623, Z    +0.000, E1   -38.580, E3 +391436.840}
SPL {X  -161.983, Y  +710.160, Z    +0.000, E1   -38.439, E3 +391446.619}
SPL {X  -161.163, Y  +713.794, Z    +0.000, E1   -38.390, E3 +391455.989}
SPL {X  -160.158, Y  +717.801, Z    +0.000, E1   -38.225, E3 +391467.119}
SPL {X  -155.870, Y  +731.575, Z    +0.000, E1   -42.661, E3 +391474.582}
SPL {X  -137.799, Y  +767.431, Z    +0.000, E1   -46.550, E3 +391531.092}
ENDSPLINE

SPLINE
SPL {X  -141.948, Y  +760.885, Z    +0.000, E1   -42.258, E3 +391563.228}
SPL {X  -160.264, Y  +717.397, Z    +0.000, E1   -24.835, E3 +391604.413}
SPL {X  -164.457, Y  +695.345, Z    +0.000, E1   -14.031, E3 +391611.355}
SPL {X  -165.312, Y  +686.072, Z    +0.000, E1    -9.096, E3 +391604.448}
SPL {X  -165.625, Y  +678.398, Z    +0.000, E1    -4.508, E3 +391602.191}
SPL {X  -165.650, Y  +672.825, Z    +0.000, E1    -0.909, E3 +391601.339}
SPL {X  -165.650, Y  +667.803, Z    +0.000, E1    +2.989, E3 +391600.799}
SPL {X  -165.650, Y  +662.773, Z    +0.000, E1    +7.549, E3 +391600.721}
SPL {X  -165.650, Y  +656.581, Z    +0.000, E1   +13.870, E3 +391598.770}
SPL {X  -165.650, Y  +648.120, Z    +0.000, E1   +22.794, E3 +391598.001}
SPL {X  -165.650, Y  +632.103, Z    +0.000, E1   +42.949, E3 +391584.959}
SPL {X  -165.650, Y  +608.448, Z    +0.000, E1   +47.265, E3 +391611.399}
SPL {X  -165.650, Y  +595.526, Z    +0.000, E1   +48.856, E3 +391625.257}
SPL {X  -165.650, Y  +568.828, Z    +0.000, E1   +48.639, E3 +391667.810}
ENDSPLINE

SPLINE
SPL {X  -165.650, Y  +586.972, Z    +0.000, E1   +40.422, E3 +391678.509}
ENDSPLINE

SPLINE
SPL {X  -165.650, Y  +585.370, Z    +0.000, E1   +38.910, E3 +391691.769}
SPL {X  -165.650, Y  +580.805, Z    +0.000, E1   +38.877, E3 +391703.391}
SPL {X  -165.650, Y  +576.923, Z    +0.000, E1   +38.908, E3 +391713.068}
SPL {X  -165.650, Y  +571.957, Z    +0.000, E1   +38.951, E3 +391725.473}
SPL {X  -165.650, Y  +566.463, Z    +0.000, E1   +38.933, E3 +391739.446}
SPL {X  -165.650, Y  +561.565, Z    +0.000, E1   +38.903, E3 +391752.019}
SPL {X  -165.650, Y  +557.881, Z    +0.000, E1   +38.850, E3 +391761.594}
SPL {X  -165.650, Y  +552.770, Z    +0.000, E1   +38.963, E3 +391774.063}
SPL {X  -165.650, Y  +548.337, Z    +0.000, E1   +38.743, E3 +391786.443}
SPL {X  -165.650, Y  +542.772, Z    +0.000, E1   +39.054, E3 +391798.821}
SPL {X  -165.650, Y  +537.647, Z    +0.000, E1   +38.838, E3 +391812.984}
SPL {X  -165.650, Y  +532.636, Z    +0.000, E1   +39.009, E3 +391824.630}
SPL {X  -165.650, Y  +528.320, Z    +0.000, E1   +38.809, E3 +391836.813}
SPL {X  -165.650, Y  +522.377, Z    +0.000, E1   +38.974, E3 +391850.933}
ENDSPLINE

SPLINE
SPL {X  -165.650, Y  +539.854, Z    +0.000, E1   +28.090, E3 +391867.550}
ENDSPLINE

SPLINE
SPL {X  -165.650, Y  +534.443, Z    +0.000, E1   +28.969, E3 +391881.601}
SPL {X  -165.650, Y  +530.452, Z    +0.000, E1   +29.664, E3 +391891.334}
SPL {X  -165.650, Y  +525.298, Z    +0.000, E1   +30.602, E3 +391903.145}
SPL {X  -165.650, Y  +518.290, Z    +0.000, E1   +31.783, E3 +391919.037}
SPL {X  -165.650, Y  +512.706, Z    +0.000, E1   +32.573, E3 +391931.871}
SPL {X  -165.650, Y  +507.785, Z    +0.000, E1   +33.438, E3 +391941.809}
SPL {X  -165.650, Y  +501.257, Z    +0.000, E1   +34.478, E3 +391955.048}
SPL {X  -165.650, Y  +495.236, Z    +0.000, E1   +35.288, E3 +391967.554}
SPL {X  -165.650, Y  +488.684, Z    +0.000, E1   +36.217, E3 +391980.451}
SPL {X  -165.650, Y  +483.157, Z    +0.000, E1   +36.957, E3 +391991.013}
SPL {X  -165.650, Y  +477.375, Z    +0.000, E1   +37.747, E3 +392001.778}
SPL {X  -165.650, Y  +469.901, Z    +0.000, E1   +38.767, E3 +392014.910}
SPL {X  -165.650, Y  +461.805, Z    +0.000, E1   +39.619, E3 +392030.253}
SPL {X  -165.650, Y  +455.681, Z    +0.000, E1   +39.641, E3 +392045.042}
SPL {X  -165.650, Y  +451.332, Z    +0.000, E1   +39.738, E3 +392055.175}
SPL {X  -165.650, Y  +448.050, Z    +0.000, E1   +39.392, E3 +392065.341}
SPL {X  -165.650, Y  +442.946, Z    +0.000, E1   +39.866, E3 +392075.115}
SPL {X  -165.650, Y  +439.091, Z    +0.000, E1   +39.674, E3 +392085.733}
SPL {X  -165.650, Y  +434.131, Z    +0.000, E1   +39.643, E3 +392098.246}
SPL {X  -165.650, Y  +428.810, Z    +0.000, E1   +39.691, E3 +392111.008}
SPL {X  -165.650, Y  +424.197, Z    +0.000, E1   +39.695, E3 +392122.367}
SPL {X  -165.650, Y  +420.220, Z    +0.000, E1   +39.526, E3 +392133.162}
SPL {X  -165.650, Y  +414.177, Z    +0.000, E1   +39.693, E3 +392147.288}
SPL {X  -165.650, Y  +407.394, Z    +0.000, E1   +39.797, E3 +392163.243}
SPL {X  -165.650, Y  +402.798, Z    +0.000, E1   +39.651, E3 +392175.365}
SPL {X  -165.650, Y  +398.253, Z    +0.000, E1   +39.688, E3 +392186.368}
SPL {X  -165.650, Y  +393.720, Z    +0.000, E1   +39.686, E3 +392197.543}
SPL {X  -165.650, Y  +389.210, Z    +0.000, E1   +39.696, E3 +392208.592}
SPL {X  -165.650, Y  +384.878, Z    +0.000, E1   +39.631, E3 +392219.669}
SPL {X  -165.650, Y  +380.529, Z    +0.000, E1   +39.528, E3 +392231.055}
SPL {X  -165.618, Y  +375.240, Z    +0.000, E1   +39.617, E3 +392243.650}
SPL {X  -165.428, Y  +369.922, Z    +0.000, E1   +39.705, E3 +392256.191}
SPL {X  -165.216, Y  +366.519, Z    +0.000, E1   +39.498, E3 +392265.758}
SPL {X  -164.790, Y  +361.646, Z    +0.000, E1   +39.684, E3 +392276.752}
SPL {X  -164.317, Y  +357.530, Z    +0.000, E1   +39.402, E3 +392288.466}
SPL {X  -163.775, Y  +353.645, Z    +0.000, E1   +39.313, E3 +392298.636}
SPL {X  -162.932, Y  +348.615, Z    +0.000, E1   +39.259, E3 +392311.400}
SPL {X  -162.143, Y  +344.596, Z    +0.000, E1   +39.019, E3 +392322.617}
SPL {X  -161.093, Y  +339.912, Z    +0.000, E1   +38.966, E3 +392334.568}
SPL {X  -159.926, Y  +335.332, Z    +0.000, E1   +38.809, E3 +392346.622}
SPL {X  -153.020, Y  +315.059, Z    +0.000, E1   +45.580, E3 +392353.353}
SPL {X  -148.632, Y  +305.368, Z    +0.000, E1   +40.700, E3 +392412.955}
SPL {X  -145.004, Y  +298.414, Z    +0.000, E1   +40.971, E3 +392437.690}
ENDSPLINE

SPLINE
SPL {X  -149.687, Y  +307.551, Z    +0.000, E1   +36.303, E3 +392473.122}
SPL {X  -158.807, Y  +331.381, Z    +0.000, E1   +26.928, E3 +392496.775}
SPL {X  -164.505, Y  +359.058, Z    +0.000, E1   +13.887, E3 +392485.537}
SPL {X  -165.494, Y  +371.321, Z    +0.000, E1    +7.176, E3 +392484.097}
SPL {X  -165.650, Y  +379.419, Z    +0.000, E1    +2.065, E3 +392481.779}
SPL {X  -165.650, Y  +383.176, Z    +0.000, E1    -0.610, E3 +392482.774}
SPL {X  -165.650, Y  +388.696, Z    +0.000, E1    -5.134, E3 +392481.050}
SPL {X  -165.650, Y  +394.663, Z    +0.000, E1   -10.843, E3 +392482.206}
SPL {X  -165.650, Y  +400.450, Z    +0.000, E1   -18.287, E3 +392473.505}
SPL {X  -165.650, Y  +409.248, Z    +0.000, E1   -26.478, E3 +392477.128}
SPL {X  -165.650, Y  +418.660, Z    +0.000, E1   -36.186, E3 +392474.604}
SPL {X  -165.650, Y  +444.260, Z    +0.000, E1   -47.328, E3 +392490.352}
SPL {X  -165.650, Y  +458.981, Z    +0.000, E1   -49.189, E3 +392505.896}
SPL {X  -165.650, Y  +493.049, Z    +0.000, E1   -51.657, E3 +392544.929}
ENDSPLINE

SPLINE
SPL {X  -165.650, Y  +468.984, Z    +0.000, E1   -41.461, E3 +392557.789}
SPL {X  -165.650, Y  +467.052, Z    +0.000, E1   -38.928, E3 +392568.404}
ENDSPLINE

SPLINE
SPL {X  -165.650, Y  +471.956, Z    +0.000, E1   -39.047, E3 +392580.055}
SPL {X  -165.650, Y  +478.019, Z    +0.000, E1   -39.139, E3 +392594.939}
SPL {X  -165.650, Y  +484.115, Z    +0.000, E1   -39.050, E3 +392610.700}
SPL {X  -165.650, Y  +488.489, Z    +0.000, E1   -39.102, E3 +392621.309}
SPL {X  -165.650, Y  +493.422, Z    +0.000, E1   -39.176, E3 +392633.455}
SPL {X  -165.650, Y  +499.941, Z    +0.000, E1   -39.068, E3 +392650.505}
SPL {X  -165.650, Y  +505.989, Z    +0.000, E1   -39.067, E3 +392665.685}
SPL {X  -165.650, Y  +512.188, Z    +0.000, E1   -39.077, E3 +392681.327}
SPL {X  -165.650, Y  +518.439, Z    +0.000, E1   -39.071, E3 +392697.052}
SPL {X  -165.650, Y  +523.032, Z    +0.000, E1   -38.966, E3 +392709.188}
SPL {X  -165.650, Y  +527.474, Z    +0.000, E1   -39.169, E3 +392719.138}
SPL {X  -165.650, Y  +532.836, Z    +0.000, E1   -39.150, E3 +392732.920}
SPL {X  -165.650, Y  +537.667, Z    +0.000, E1   -38.986, E3 +392745.865}
SPL {X  -165.650, Y  +542.804, Z    +0.000, E1   -39.141, E3 +392758.050}
SPL {X  -165.650, Y  +547.280, Z    +0.000, E1   -38.965, E3 +392770.194}
SPL {X  -165.650, Y  +551.666, Z    +0.000, E1   -39.102, E3 +392780.512}
SPL {X  -165.650, Y  +557.612, Z    +0.000, E1   -39.166, E3 +392795.159}
SPL {X  -165.650, Y  +562.850, Z    +0.000, E1   -38.959, E3 +392809.517}
SPL {X  -165.650, Y  +568.257, Z    +0.000, E1   -39.077, E3 +392822.472}
SPL {X  -165.650, Y  +573.200, Z    +0.000, E1   -39.061, E3 +392835.007}
SPL {X  -165.650, Y  +578.240, Z    +0.000, E1   -39.117, E3 +392847.348}
SPL {X  -165.650, Y  +582.804, Z    +0.000, E1   -39.080, E3 +392859.055}
SPL {X  -165.650, Y  +587.640, Z    +0.000, E1   -39.069, E3 +392871.312}
SPL {X  -165.650, Y  +593.610, Z    +0.000, E1   -39.204, E3 +392885.586}
SPL {X  -165.650, Y  +599.021, Z    +0.000, E1   -38.950, E3 +392900.735}
SPL {X  -165.650, Y  +604.635, Z    +0.000, E1   -39.163, E3 +392913.512}
SPL {X  -165.650, Y  +608.365, Z    +0.000, E1   -39.063, E3 +392923.502}
SPL {X  -165.650, Y  +613.618, Z    +0.000, E1   -39.137, E3 +392936.366}
SPL {X  -165.650, Y  +619.584, Z    +0.000, E1   -39.045, E3 +392952.003}
SPL {X  -165.650, Y  +625.662, Z    +0.000, E1   -39.189, E3 +392966.317}
SPL {X  -165.650, Y  +629.982, Z    +0.000, E1   -39.063, E3 +392977.919}
SPL {X  -165.650, Y  +634.317, Z    +0.000, E1   -39.239, E3 +392987.709}
SPL {X  -165.650, Y  +639.215, Z    +0.000, E1   -39.074, E3 +393001.234}
SPL {X  -165.650, Y  +645.443, Z    +0.000, E1   -39.032, E3 +393017.101}
SPL {X  -165.650, Y  +651.452, Z    +0.000, E1   -39.128, E3 +393031.671}
SPL {X  -165.650, Y  +656.920, Z    +0.000, E1   -39.120, E3 +393045.448}
SPL {X  -165.650, Y  +662.945, Z    +0.000, E1   -39.141, E3 +393060.553}
SPL {X  -165.650, Y  +668.296, Z    +0.000, E1   -39.077, E3 +393074.278}
SPL {X  -165.650, Y  +674.193, Z    +0.000, E1   -39.034, E3 +393089.620}
SPL {X  -165.521, Y  +682.029, Z    +0.000, E1   -39.160, E3 +393108.588}
SPL {X  -165.139, Y  +688.497, Z    +0.000, E1   -39.013, E3 +393125.658}
SPL {X  -164.582, Y  +694.282, Z    +0.000, E1   -38.975, E3 +393140.406}
SPL {X  -163.926, Y  +699.336, Z    +0.000, E1   -38.767, E3 +393154.384}
SPL {X  -162.937, Y  +705.358, Z    +0.000, E1   -38.703, E3 +393169.968}
SPL {X  -161.983, Y  +710.160, Z    +0.000, E1   -38.439, E3 +393183.462}
SPL {X  -160.874, Y  +714.989, Z    +0.000, E1   -38.205, E3 +393197.123}
SPL {X  -158.364, Y  +724.087, Z    +0.000, E1   -39.961, E3 +393209.329}
SPL {X  -138.706, Y  +766.057, Z    +0.000, E1   -46.957, E3 +393260.320}
ENDSPLINE

SPLINE
SPL {X  -141.948, Y  +760.885, Z    +0.000, E1   -42.258, E3 +393300.070}
SPL {X  -160.264, Y  +717.397, Z    +0.000, E1   -24.835, E3 +393341.255}
SPL {X  -164.457, Y  +695.345, Z    +0.000, E1   -14.031, E3 +393348.197}
SPL {X  -165.312, Y  +686.072, Z    +0.000, E1    -9.096, E3 +393341.290}
SPL {X  -165.625, Y  +678.398, Z    +0.000, E1    -4.508, E3 +393339.033}
SPL {X  -165.650, Y  +672.825, Z    +0.000, E1    -0.909, E3 +393338.181}
SPL {X  -165.650, Y  +667.803, Z    +0.000, E1    +2.989, E3 +393337.641}
SPL {X  -165.650, Y  +662.773, Z    +0.000, E1    +7.549, E3 +393337.563}
SPL {X  -165.650, Y  +656.581, Z    +0.000, E1   +13.870, E3 +393335.612}
SPL {X  -165.650, Y  +648.120, Z    +0.000, E1   +22.794, E3 +393334.843}
SPL {X  -165.650, Y  +632.103, Z    +0.000, E1   +42.949, E3 +393321.801}
SPL {X  -165.650, Y  +608.448, Z    +0.000, E1   +47.265, E3 +393348.241}
SPL {X  -165.650, Y  +595.526, Z    +0.000, E1   +48.856, E3 +393362.099}
SPL {X  -165.650, Y  +568.828, Z    +0.000, E1   +48.639, E3 +393404.652}
ENDSPLINE

SPLINE
SPL {X  -165.650, Y  +587.144, Z    +0.000, E1   +39.840, E3 +393418.685}
ENDSPLINE

SPLINE
SPL {X  -165.650, Y  +582.480, Z    +0.000, E1   +38.929, E3 +393435.881}
SPL {X  -165.650, Y  +576.923, Z    +0.000, E1   +38.908, E3 +393449.910}
SPL {X  -165.650, Y  +570.800, Z    +0.000, E1   +39.001, E3 +393465.085}
SPL {X  -165.650, Y  +565.658, Z    +0.000, E1   +38.868, E3 +393478.623}
SPL {X  -165.650, Y  +561.565, Z    +0.000, E1   +38.903, E3 +393488.861}
SPL {X  -165.650, Y  +555.731, Z    +0.000, E1   +38.913, E3 +393503.718}
SPL {X  -165.650, Y  +549.409, Z    +0.000, E1   +38.884, E3 +393519.868}
SPL {X  -165.650, Y  +544.480, Z    +0.000, E1   +38.998, E3 +393531.531}
SPL {X  -165.650, Y  +541.194, Z    +0.000, E1   +39.037, E3 +393539.580}
SPL {X  -165.650, Y  +537.647, Z    +0.000, E1   +38.838, E3 +393549.826}
SPL {X  -165.650, Y  +532.636, Z    +0.000, E1   +39.009, E3 +393561.472}
SPL {X  -165.650, Y  +528.320, Z    +0.000, E1   +38.809, E3 +393573.655}
SPL {X  -165.650, Y  +522.377, Z    +0.000, E1   +38.974, E3 +393587.775}
ENDSPLINE

SPLINE
SPL {X  -165.650, Y  +539.854, Z    +0.000, E1   +28.090, E3 +393604.392}
ENDSPLINE

SPLINE
SPL {X  -165.650, Y  +534.443, Z    +0.000, E1   +28.969, E3 +393618.443}
SPL {X  -165.650, Y  +530.452, Z    +0.000, E1   +29.664, E3 +393628.176}
SPL {X  -165.650, Y  +523.712, Z    +0.000, E1   +30.911, E3 +393643.458}
SPL {X  -165.650, Y  +516.975, Z    +0.000, E1   +31.942, E3 +393659.052}
SPL {X  -165.650, Y  +512.706, Z    +0.000, E1   +32.573, E3 +393668.713}
SPL {X  -165.650, Y  +507.785, Z    +0.000, E1   +33.438, E3 +393678.651}
SPL {X  -165.650, Y  +502.877, Z    +0.000, E1   +34.230, E3 +393688.539}
SPL {X  -165.650, Y  +496.704, Z    +0.000, E1   +35.113, E3 +393701.332}
SPL {X  -165.650, Y  +488.684, Z    +0.000, E1   +36.217, E3 +393717.293}
SPL {X  -165.650, Y  +483.157, Z    +0.000, E1   +36.957, E3 +393727.855}
SPL {X  -165.650, Y  +477.375, Z    +0.000, E1   +37.747, E3 +393738.620}
SPL {X  -165.650, Y  +469.901, Z    +0.000, E1   +38.767, E3 +393751.752}
SPL {X  -165.650, Y  +465.276, Z    +0.000, E1   +39.067, E3 +393761.629}
SPL {X  -165.650, Y  +459.623, Z    +0.000, E1   +39.919, E3 +393770.565}
SPL {X  -165.650, Y  +455.681, Z    +0.000, E1   +39.641, E3 +393781.885}
SPL {X  -165.650, Y  +451.332, Z    +0.000, E1   +39.738, E3 +393792.017}
SPL {X  -165.650, Y  +448.050, Z    +0.000, E1   +39.392, E3 +393802.183}
SPL {X  -165.650, Y  +442.946, Z    +0.000, E1   +39.866, E3 +393811.957}
SPL {X  -165.650, Y  +439.091, Z    +0.000, E1   +39.674, E3 +393822.575}
SPL {X  -165.650, Y  +434.131, Z    +0.000, E1   +39.643, E3 +393835.088}
SPL {X  -165.650, Y  +428.810, Z    +0.000, E1   +39.691, E3 +393847.850}
SPL {X  -165.650, Y  +424.197, Z    +0.000, E1   +39.695, E3 +393859.209}
SPL {X  -165.650, Y  +420.220, Z    +0.000, E1   +39.526, E3 +393870.004}
SPL {X  -165.650, Y  +414.177, Z    +0.000, E1   +39.693, E3 +393884.131}
SPL {X  -165.650, Y  +407.394, Z    +0.000, E1   +39.797, E3 +393900.085}
SPL {X  -165.650, Y  +402.798, Z    +0.000, E1   +39.651, E3 +393912.207}
SPL {X  -165.650, Y  +398.253, Z    +0.000, E1   +39.688, E3 +393923.210}
SPL {X  -165.650, Y  +393.720, Z    +0.000, E1   +39.686, E3 +393934.385}
SPL {X  -165.650, Y  +389.210, Z    +0.000, E1   +39.696, E3 +393945.434}
SPL {X  -165.650, Y  +384.878, Z    +0.000, E1   +39.631, E3 +393956.511}
SPL {X  -165.650, Y  +380.529, Z    +0.000, E1   +39.528, E3 +393967.897}
SPL {X  -165.618, Y  +375.240, Z    +0.000, E1   +39.617, E3 +393980.492}
SPL {X  -165.428, Y  +369.922, Z    +0.000, E1   +39.705, E3 +393993.033}
SPL {X  -165.216, Y  +366.519, Z    +0.000, E1   +39.498, E3 +394002.600}
SPL {X  -164.790, Y  +361.646, Z    +0.000, E1   +39.684, E3 +394013.594}
SPL {X  -164.317, Y  +357.530, Z    +0.000, E1   +39.402, E3 +394025.308}
SPL {X  -163.775, Y  +353.645, Z    +0.000, E1   +39.313, E3 +394035.478}
SPL {X  -163.109, Y  +349.595, Z    +0.000, E1   +39.290, E3 +394045.540}
SPL {X  -162.309, Y  +345.398, Z    +0.000, E1   +39.085, E3 +394057.204}
SPL {X  -161.467, Y  +341.510, Z    +0.000, E1   +38.980, E3 +394067.249}
SPL {X  -160.812, Y  +338.758, Z    +0.000, E1   +38.898, E3 +394074.506}
SPL {X  -159.926, Y  +335.332, Z    +0.000, E1   +38.809, E3 +394083.464}
SPL {X  -153.020, Y  +315.059, Z    +0.000, E1   +45.580, E3 +394090.195}
SPL {X  -148.632, Y  +305.368, Z    +0.000, E1   +40.700, E3 +394149.797}
SPL {X  -145.004, Y  +298.414, Z    +0.000, E1   +40.971, E3 +394174.532}
ENDSPLINE

SPLINE
SPL {X  -149.687, Y  +307.551, Z    +0.000, E1   +36.303, E3 +394209.964}
SPL {X  -158.807, Y  +331.381, Z    +0.000, E1   +26.928, E3 +394233.617}
SPL {X  -164.505, Y  +359.058, Z    +0.000, E1   +13.887, E3 +394222.379}
SPL {X  -165.494, Y  +371.321, Z    +0.000, E1    +7.176, E3 +394220.939}
SPL {X  -165.650, Y  +379.419, Z    +0.000, E1    +2.065, E3 +394218.621}
SPL {X  -165.650, Y  +383.176, Z    +0.000, E1    -0.610, E3 +394219.616}
SPL {X  -165.650, Y  +387.435, Z    +0.000, E1    -4.104, E3 +394217.976}
SPL {X  -165.650, Y  +393.422, Z    +0.000, E1    -9.605, E3 +394218.533}
SPL {X  -165.650, Y  +400.450, Z    +0.000, E1   -18.287, E3 +394210.348}
SPL {X  -165.650, Y  +409.248, Z    +0.000, E1   -26.478, E3 +394213.970}
SPL {X  -165.650, Y  +418.660, Z    +0.000, E1   -36.186, E3 +394211.446}
SPL {X  -165.650, Y  +444.260, Z    +0.000, E1   -47.328, E3 +394227.194}
SPL {X  -165.650, Y  +458.981, Z    +0.000, E1   -49.189, E3 +394242.738}
SPL {X  -165.650, Y  +493.049, Z    +0.000, E1   -51.657, E3 +394281.771}
ENDSPLINE

SPLINE
SPL {X  -165.650, Y  +468.984, Z    +0.000, E1   -41.461, E3 +394294.631}
SPL {X  -165.650, Y  +467.052, Z    +0.000, E1   -38.928, E3 +394305.246}
ENDSPLINE

SPLINE
SPL {X  -165.650, Y  +471.956, Z    +0.000, E1   -39.047, E3 +394316.897}
SPL {X  -165.650, Y  +476.270, Z    +0.000, E1   -39.142, E3 +394327.153}
SPL {X  -165.650, Y  +480.876, Z    +0.000, E1   -39.050, E3 +394339.435}
SPL {X  -165.650, Y  +487.054, Z    +0.000, E1   -39.118, E3 +394354.574}
SPL {X  -165.650, Y  +491.785, Z    +0.000, E1   -39.157, E3 +394366.123}
SPL {X  -165.650, Y  +496.519, Z    +0.000, E1   -39.062, E3 +394378.738}
SPL {X  -165.650, Y  +501.480, Z    +0.000, E1   -39.099, E3 +394390.894}
SPL {X  -165.650, Y  +505.989, Z    +0.000, E1   -39.067, E3 +394402.527}
SPL {X  -165.650, Y  +512.188, Z    +0.000, E1   -39.077, E3 +394418.170}
SPL {X  -165.650, Y  +518.439, Z    +0.000, E1   -39.071, E3 +394433.895}
SPL {X  -165.650, Y  +523.032, Z    +0.000, E1   -38.966, E3 +394446.030}
SPL {X  -165.650, Y  +527.474, Z    +0.000, E1   -39.169, E3 +394455.980}
SPL {X  -165.650, Y  +532.836, Z    +0.000, E1   -39.150, E3 +394469.763}
SPL {X  -165.650, Y  +539.651, Z    +0.000, E1   -39.087, E3 +394487.280}
SPL {X  -165.650, Y  +544.603, Z    +0.000, E1   -39.103, E3 +394499.456}
SPL {X  -165.650, Y  +547.280, Z    +0.000, E1   -38.965, E3 +394507.036}
SPL {X  -165.650, Y  +551.666, Z    +0.000, E1   -39.102, E3 +394517.354}
SPL {X  -165.650, Y  +557.612, Z    +0.000, E1   -39.166, E3 +394532.001}
SPL {X  -165.650, Y  +562.850, Z    +0.000, E1   -38.959, E3 +394546.359}
SPL {X  -165.650, Y  +568.257, Z    +0.000, E1   -39.077, E3 +394559.315}
SPL {X  -165.650, Y  +573.200, Z    +0.000, E1   -39.061, E3 +394571.849}
SPL {X  -165.650, Y  +578.240, Z    +0.000, E1   -39.117, E3 +394584.190}
SPL {X  -165.650, Y  +582.804, Z    +0.000, E1   -39.080, E3 +394595.897}
SPL {X  -165.650, Y  +587.640, Z    +0.000, E1   -39.069, E3 +394608.154}
SPL {X  -165.650, Y  +592.685, Z    +0.000, E1   -39.263, E3 +394619.619}
SPL {X  -165.650, Y  +596.539, Z    +0.000, E1   -39.049, E3 +394630.608}
SPL {X  -165.650, Y  +599.973, Z    +0.000, E1   -38.814, E3 +394640.661}
SPL {X  -165.650, Y  +604.635, Z    +0.000, E1   -39.163, E3 +394650.354}
SPL {X  -165.650, Y  +608.365, Z    +0.000, E1   -39.063, E3 +394660.344}
SPL {X  -165.650, Y  +612.142, Z    +0.000, E1   -39.023, E3 +394670.074}
SPL {X  -165.650, Y  +616.635, Z    +0.000, E1   -39.260, E3 +394679.962}
SPL {X  -165.650, Y  +620.299, Z    +0.000, E1   -38.904, E3 +394691.348}
SPL {X  -165.650, Y  +625.662, Z    +0.000, E1   -39.189, E3 +394703.159}
SPL {X  -165.650, Y  +629.982, Z    +0.000, E1   -39.063, E3 +394714.761}
SPL {X  -165.650, Y  +635.019, Z    +0.000, E1   -39.106, E3 +394727.243}
SPL {X  -165.650, Y  +641.706, Z    +0.000, E1   -39.097, E3 +394744.310}
SPL {X  -165.650, Y  +648.294, Z    +0.000, E1   -39.142, E3 +394760.432}
SPL {X  -165.650, Y  +652.477, Z    +0.000, E1   -39.068, E3 +394771.335}
SPL {X  -165.650, Y  +656.920, Z    +0.000, E1   -39.120, E3 +394782.290}
SPL {X  -165.650, Y  +661.125, Z    +0.000, E1   -39.092, E3 +394792.938}
SPL {X  -165.650, Y  +664.437, Z    +0.000, E1   -39.114, E3 +394801.147}
SPL {X  -165.650, Y  +668.296, Z    +0.000, E1   -39.077, E3 +394811.120}
SPL {X  -165.650, Y  +674.193, Z    +0.000, E1   -39.034, E3 +394826.462}
SPL {X  -165.521, Y  +682.029, Z    +0.000, E1   -39.160, E3 +394845.430}
SPL {X  -165.241, Y  +687.126, Z    +0.000, E1   -39.221, E3 +394857.591}
SPL {X  -165.072, Y  +689.330, Z    +0.000, E1   -38.812, E3 +394865.640}
SPL {X  -164.582, Y  +694.282, Z    +0.000, E1   -38.975, E3 +394877.248}
SPL {X  -163.926, Y  +699.336, Z    +0.000, E1   -38.767, E3 +394891.226}
SPL {X  -163.214, Y  +703.806, Z    +0.000, E1   -38.755, E3 +394902.411}
SPL {X  -162.700, Y  +706.623, Z    +0.000, E1   -38.580, E3 +394910.524}
SPL {X  -161.983, Y  +710.160, Z    +0.000, E1   -38.439, E3 +394920.304}
SPL {X  -161.163, Y  +713.794, Z    +0.000, E1   -38.390, E3 +394929.673}
SPL {X  -160.616, Y  +716.027, Z    +0.000, E1   -37.944, E3 +394937.876}
SPL {X  -158.364, Y  +724.087, Z    +0.000, E1   -39.961, E3 +394946.171}
SPL {X  -138.706, Y  +766.057, Z    +0.000, E1   -46.957, E3 +394997.162}
ENDSPLINE

SPLINE
SPL {X  -141.948, Y  +760.885, Z    +0.000, E1   -42.258, E3 +395036.913}
SPL {X  -152.484, Y  +740.219, Z    +0.000, E1   -33.928, E3 +395074.066}
SPL {X  -161.203, Y  +713.624, Z    +0.000, E1   -23.097, E3 +395078.482}
SPL {X  -164.762, Y  +692.628, Z    +0.000, E1   -12.660, E3 +395081.350}
SPL {X  -165.481, Y  +682.990, Z    +0.000, E1    -7.255, E3 +395078.194}
SPL {X  -165.649, Y  +676.021, Z    +0.000, E1    -3.061, E3 +395075.561}
SPL {X  -165.650, Y  +670.589, Z    +0.000, E1    +0.778, E3 +395074.799}
SPL {X  -165.650, Y  +666.842, Z    +0.000, E1    +3.871, E3 +395074.260}
SPL {X  -165.650, Y  +662.773, Z    +0.000, E1    +7.549, E3 +395074.405}
SPL {X  -165.650, Y  +656.581, Z    +0.000, E1   +13.870, E3 +395072.454}
SPL {X  -165.650, Y  +648.120, Z    +0.000, E1   +22.794, E3 +395071.685}
SPL {X  -165.650, Y  +632.103, Z    +0.000, E1   +42.949, E3 +395058.643}
SPL {X  -165.650, Y  +609.948, Z    +0.000, E1   +49.636, E3 +395076.070}
SPL {X  -165.650, Y  +601.895, Z    +0.000, E1   +47.595, E3 +395093.740}
SPL {X  -165.650, Y  +568.828, Z    +0.000, E1   +48.639, E3 +395141.494}
ENDSPLINE

SPLINE
SPL {X  -165.650, Y  +586.972, Z    +0.000, E1   +40.422, E3 +395152.193}
ENDSPLINE

SPLINE
SPL {X  -165.650, Y  +585.370, Z    +0.000, E1   +38.910, E3 +395165.453}
SPL {X  -165.650, Y  +580.805, Z    +0.000, E1   +38.877, E3 +395177.075}
SPL {X  -165.650, Y  +575.679, Z    +0.000, E1   +38.947, E3 +395189.798}
SPL {X  -165.650, Y  +569.616, Z    +0.000, E1   +38.966, E3 +395204.956}
SPL {X  -165.650, Y  +564.364, Z    +0.000, E1   +38.909, E3 +395218.609}
SPL {X  -165.650, Y  +559.065, Z    +0.000, E1   +38.883, E3 +395232.187}
SPL {X  -165.650, Y  +552.770, Z    +0.000, E1   +38.963, E3 +395247.748}
SPL {X  -165.650, Y  +548.337, Z    +0.000, E1   +38.743, E3 +395260.127}
SPL {X  -165.650, Y  +542.772, Z    +0.000, E1   +39.054, E3 +395272.505}
SPL {X  -165.650, Y  +537.647, Z    +0.000, E1   +38.838, E3 +395286.668}
SPL {X  -165.650, Y  +532.636, Z    +0.000, E1   +39.009, E3 +395298.314}
SPL {X  -165.650, Y  +528.320, Z    +0.000, E1   +38.809, E3 +395310.497}
SPL {X  -165.650, Y  +522.377, Z    +0.000, E1   +38.974, E3 +395324.617}
ENDSPLINE

SPLINE
SPL {X  -165.650, Y  +541.168, Z    +0.000, E1   +27.957, E3 +395336.957}
ENDSPLINE

SPLINE
SPL {X  -165.650, Y  +536.052, Z    +0.000, E1   +28.653, E3 +395351.592}
SPL {X  -165.650, Y  +530.452, Z    +0.000, E1   +29.664, E3 +395365.019}
SPL {X  -165.650, Y  +523.712, Z    +0.000, E1   +30.911, E3 +395380.300}
SPL {X  -165.650, Y  +516.975, Z    +0.000, E1   +31.942, E3 +395395.894}
SPL {X  -165.650, Y  +512.706, Z    +0.000, E1   +32.573, E3 +395405.555}
SPL {X  -165.650, Y  +507.785, Z    +0.000, E1   +33.438, E3 +395415.493}
SPL {X  -165.650, Y  +501.257, Z    +0.000, E1   +34.478, E3 +395428.732}
SPL {X  -165.650, Y  +495.236, Z    +0.000, E1   +35.288, E3 +395441.238}
SPL {X  -165.650, Y  +488.684, Z    +0.000, E1   +36.217, E3 +395454.135}
SPL {X  -165.650, Y  +481.130, Z    +0.000, E1   +37.251, E3 +395468.444}
SPL {X  -165.650, Y  +475.455, Z    +0.000, E1   +37.964, E3 +395479.100}
SPL {X  -165.650, Y  +469.901, Z    +0.000, E1   +38.767, E3 +395488.594}
SPL {X  -165.650, Y  +465.276, Z    +0.000, E1   +39.067, E3 +395498.471}
SPL {X  -165.650, Y  +459.623, Z    +0.000, E1   +39.919, E3 +395507.407}
SPL {X  -165.650, Y  +455.681, Z    +0.000, E1   +39.641, E3 +395518.727}
SPL {X  -165.650, Y  +451.332, Z    +0.000, E1   +39.738, E3 +395528.859}
SPL {X  -165.650, Y  +448.050, Z    +0.000, E1   +39.392, E3 +395539.025}
SPL {X  -165.650, Y  +442.946, Z    +0.000, E1   +39.866, E3 +395548.799}
SPL {X  -165.650, Y  +439.091, Z    +0.000, E1   +39.674, E3 +395559.417}
SPL {X  -165.650, Y  +434.131, Z    +0.000, E1   +39.643, E3 +395571.930}
SPL {X  -165.650, Y  +428.810, Z    +0.000, E1   +39.691, E3 +395584.692}
SPL {X  -165.650, Y  +424.197, Z    +0.000, E1   +39.695, E3 +395596.051}
SPL {X  -165.650, Y  +420.220, Z    +0.000, E1   +39.526, E3 +395606.846}
SPL {X  -165.650, Y  +414.177, Z    +0.000, E1   +39.693, E3 +395620.973}
SPL {X  -165.650, Y  +407.394, Z    +0.000, E1   +39.797, E3 +395636.927}
SPL {X  -165.650, Y  +402.798, Z    +0.000, E1   +39.651, E3 +395649.049}
SPL {X  -165.650, Y  +398.253, Z    +0.000, E1   +39.688, E3 +395660.052}
SPL {X  -165.650, Y  +393.720, Z    +0.000, E1   +39.686, E3 +395671.227}
SPL {X  -165.650, Y  +389.210, Z    +0.000, E1   +39.696, E3 +395682.276}
SPL {X  -165.650, Y  +384.878, Z    +0.000, E1   +39.631, E3 +395693.353}
SPL {X  -165.650, Y  +380.529, Z    +0.000, E1   +39.528, E3 +395704.739}
SPL {X  -165.618, Y  +375.240, Z    +0.000, E1   +39.617, E3 +395717.334}
SPL {X  -165.428, Y  +369.922, Z    +0.000, E1   +39.705, E3 +395729.875}
SPL {X  -165.216, Y  +366.519, Z    +0.000, E1   +39.498, E3 +395739.442}
SPL {X  -164.790, Y  +361.646, Z    +0.000, E1   +39.684, E3 +395750.436}
SPL {X  -164.317, Y  +357.530, Z    +0.000, E1   +39.402, E3 +395762.150}
SPL {X  -163.775, Y  +353.645, Z    +0.000, E1   +39.313, E3 +395772.320}
SPL {X  -163.109, Y  +349.595, Z    +0.000, E1   +39.290, E3 +395782.382}
SPL {X  -162.309, Y  +345.398, Z    +0.000, E1   +39.085, E3 +395794.046}
SPL {X  -161.467, Y  +341.510, Z    +0.000, E1   +38.980, E3 +395804.091}
SPL {X  -160.812, Y  +338.758, Z    +0.000, E1   +38.898, E3 +395811.348}
SPL {X  -159.926, Y  +335.332, Z    +0.000, E1   +38.809, E3 +395820.306}
SPL {X  -153.020, Y  +315.059, Z    +0.000, E1   +45.580, E3 +395827.037}
SPL {X  -148.632, Y  +305.368, Z    +0.000, E1   +40.700, E3 +395886.639}
SPL {X  -145.004, Y  +298.414, Z    +0.000, E1   +40.971, E3 +395911.374}
ENDSPLINE

SPLINE
SPL {X  -149.687, Y  +307.551, Z    +0.000, E1   +36.303, E3 +395946.807}
SPL {X  -158.807, Y  +331.381, Z    +0.000, E1   +26.928, E3 +395970.459}
SPL {X  -164.505, Y  +359.058, Z    +0.000, E1   +13.887, E3 +395959.221}
SPL {X  -165.334, Y  +368.271, Z    +0.000, E1    +8.886, E3 +395957.059}
SPL {X  -165.596, Y  +374.277, Z    +0.000, E1    +5.306, E3 +395958.441}
SPL {X  -165.650, Y  +379.419, Z    +0.000, E1    +2.065, E3 +395955.463}
SPL {X  -165.650, Y  +383.176, Z    +0.000, E1    -0.610, E3 +395956.458}
SPL {X  -165.650, Y  +387.435, Z    +0.000, E1    -4.104, E3 +395954.818}
SPL {X  -165.650, Y  +393.422, Z    +0.000, E1    -9.605, E3 +395955.375}
SPL {X  -165.650, Y  +400.450, Z    +0.000, E1   -18.287, E3 +395947.190}
SPL {X  -165.650, Y  +409.248, Z    +0.000, E1   -26.478, E3 +395950.812}
SPL {X  -165.650, Y  +418.660, Z    +0.000, E1   -36.186, E3 +395948.289}
SPL {X  -165.650, Y  +444.260, Z    +0.000, E1   -47.328, E3 +395964.036}
SPL {X  -165.650, Y  +458.981, Z    +0.000, E1   -49.189, E3 +395979.580}
SPL {X  -165.650, Y  +493.049, Z    +0.000, E1   -51.657, E3 +396018.613}
ENDSPLINE

SPLINE
SPL {X  -165.650, Y  +468.984, Z    +0.000, E1   -41.461, E3 +396031.473}
SPL {X  -165.650, Y  +467.052, Z    +0.000, E1   -38.928, E3 +396042.088}
ENDSPLINE

SPLINE
SPL {X  -165.650, Y  +471.956, Z    +0.000, E1   -39.047, E3 +396053.739}
SPL {X  -165.650, Y  +478.019, Z    +0.000, E1   -39.139, E3 +396068.623}
SPL {X  -165.650, Y  +484.115, Z    +0.000, E1   -39.050, E3 +396084.385}
SPL {X  -165.650, Y  +490.374, Z    +0.000, E1   -39.169, E3 +396099.504}
SPL {X  -165.650, Y  +496.519, Z    +0.000, E1   -39.062, E3 +396115.580}
SPL {X  -165.650, Y  +502.351, Z    +0.000, E1   -39.056, E3 +396130.302}
SPL {X  -165.650, Y  +508.180, Z    +0.000, E1   -39.157, E3 +396144.368}
SPL {X  -165.650, Y  +514.341, Z    +0.000, E1   -39.047, E3 +396160.620}
SPL {X  -165.650, Y  +521.541, Z    +0.000, E1   -39.052, E3 +396178.804}
SPL {X  -165.650, Y  +528.401, Z    +0.000, E1   -39.135, E3 +396195.473}
SPL {X  -165.650, Y  +533.857, Z    +0.000, E1   -39.163, E3 +396208.978}
SPL {X  -165.650, Y  +539.651, Z    +0.000, E1   -39.087, E3 +396224.122}
SPL {X  -165.650, Y  +546.018, Z    +0.000, E1   -39.065, E3 +396240.247}
SPL {X  -165.650, Y  +551.666, Z    +0.000, E1   -39.102, E3 +396254.197}
SPL {X  -165.650, Y  +555.880, Z    +0.000, E1   -39.094, E3 +396264.768}
SPL {X  -165.650, Y  +559.255, Z    +0.000, E1   -39.167, E3 +396272.804}
SPL {X  -165.650, Y  +562.850, Z    +0.000, E1   -38.959, E3 +396283.201}
SPL {X  -165.650, Y  +568.257, Z    +0.000, E1   -39.077, E3 +396296.157}
SPL {X  -165.650, Y  +573.200, Z    +0.000, E1   -39.061, E3 +396308.691}
SPL {X  -165.650, Y  +578.240, Z    +0.000, E1   -39.117, E3 +396321.032}
SPL {X  -165.650, Y  +582.804, Z    +0.000, E1   -39.080, E3 +396332.740}
SPL {X  -165.650, Y  +587.640, Z    +0.000, E1   -39.069, E3 +396344.996}
SPL {X  -165.650, Y  +592.685, Z    +0.000, E1   -39.263, E3 +396356.461}
SPL {X  -165.650, Y  +596.539, Z    +0.000, E1   -39.049, E3 +396367.450}
SPL {X  -165.650, Y  +599.973, Z    +0.000, E1   -38.814, E3 +396377.503}
SPL {X  -165.650, Y  +604.635, Z    +0.000, E1   -39.163, E3 +396387.196}
SPL {X  -165.650, Y  +608.365, Z    +0.000, E1   -39.063, E3 +396397.186}
SPL {X  -165.650, Y  +612.142, Z    +0.000, E1   -39.023, E3 +396406.916}
SPL {X  -165.650, Y  +616.635, Z    +0.000, E1   -39.260, E3 +396416.804}
SPL {X  -165.650, Y  +620.299, Z    +0.000, E1   -38.904, E3 +396428.190}
SPL {X  -165.650, Y  +625.662, Z    +0.000, E1   -39.189, E3 +396440.001}
SPL {X  -165.650, Y  +629.982, Z    +0.000, E1   -39.063, E3 +396451.603}
SPL {X  -165.650, Y  +635.019, Z    +0.000, E1   -39.106, E3 +396464.085}
SPL {X  -165.650, Y  +641.706, Z    +0.000, E1   -39.097, E3 +396481.152}
SPL {X  -165.650, Y  +648.294, Z    +0.000, E1   -39.142, E3 +396497.274}
SPL {X  -165.650, Y  +652.477, Z    +0.000, E1   -39.068, E3 +396508.177}
SPL {X  -165.650, Y  +656.920, Z    +0.000, E1   -39.120, E3 +396519.132}
SPL {X  -165.650, Y  +662.945, Z    +0.000, E1   -39.141, E3 +396534.237}
SPL {X  -165.650, Y  +668.296, Z    +0.000, E1   -39.077, E3 +396547.962}
SPL {X  -165.650, Y  +673.138, Z    +0.000, E1   -39.196, E3 +396559.418}
SPL {X  -165.640, Y  +677.281, Z    +0.000, E1   -38.803, E3 +396572.306}
SPL {X  -165.389, Y  +684.794, Z    +0.000, E1   -39.261, E3 +396588.617}
SPL {X  -164.948, Y  +690.736, Z    +0.000, E1   -38.951, E3 +396605.286}
SPL {X  -164.363, Y  +696.109, Z    +0.000, E1   -38.853, E3 +396619.376}
SPL {X  -163.795, Y  +700.218, Z    +0.000, E1   -38.698, E3 +396630.584}
SPL {X  -162.937, Y  +705.358, Z    +0.000, E1   -38.703, E3 +396643.652}
SPL {X  -161.983, Y  +710.160, Z    +0.000, E1   -38.439, E3 +396657.146}
SPL {X  -160.874, Y  +714.989, Z    +0.000, E1   -38.205, E3 +396670.807}
SPL {X  -158.364, Y  +724.087, Z    +0.000, E1   -39.961, E3 +396683.013}
SPL {X  -138.706, Y  +766.057, Z    +0.000, E1   -46.957, E3 +396734.004}
ENDSPLINE

SPLINE
SPL {X  -141.948, Y  +760.885, Z    +0.000, E1   -42.258, E3 +396773.755}
SPL {X  -160.264, Y  +717.397, Z    +0.000, E1   -24.835, E3 +396814.939}
SPL {X  -164.762, Y  +692.628, Z    +0.000, E1   -12.660, E3 +396818.192}
SPL {X  -165.581, Y  +680.274, Z    +0.000, E1    -5.699, E3 +396813.676}
SPL {X  -165.650, Y  +674.578, Z    +0.000, E1    -2.045, E3 +396812.204}
SPL {X  -165.650, Y  +670.589, Z    +0.000, E1    +0.778, E3 +396811.641}
SPL {X  -165.650, Y  +666.842, Z    +0.000, E1    +3.871, E3 +396811.102}
SPL {X  -165.650, Y  +661.513, Z    +0.000, E1    +8.695, E3 +396811.010}
SPL {X  -165.650, Y  +654.973, Z    +0.000, E1   +15.752, E3 +396808.416}
SPL {X  -165.650, Y  +648.120, Z    +0.000, E1   +22.794, E3 +396808.527}
SPL {X  -165.650, Y  +632.103, Z    +0.000, E1   +42.949, E3 +396795.485}
SPL {X  -165.650, Y  +609.948, Z    +0.000, E1   +49.636, E3 +396812.912}
SPL {X  -165.650, Y  +601.895, Z    +0.000, E1   +47.595, E3 +396830.582}
SPL {X  -165.650, Y  +568.828, Z    +0.000, E1   +48.639, E3 +396878.337}
ENDSPLINE

SPLINE
SPL {X  -165.650, Y  +587.144, Z    +0.000, E1   +39.840, E3 +396892.369}
ENDSPLINE

SPLINE
SPL {X  -165.650, Y  +582.480, Z    +0.000, E1   +38.929, E3 +396909.565}
SPL {X  -165.650, Y  +576.923, Z    +0.000, E1   +38.908, E3 +396923.594}
SPL {X  -165.650, Y  +571.957, Z    +0.000, E1   +38.951, E3 +396935.999}
SPL {X  -165.650, Y  +566.463, Z    +0.000, E1   +38.933, E3 +396949.972}
SPL {X  -165.650, Y  +560.094, Z    +0.000, E1   +38.931, E3 +396966.293}
SPL {X  -165.650, Y  +554.358, Z    +0.000, E1   +38.887, E3 +396980.871}
SPL {X  -165.650, Y  +549.409, Z    +0.000, E1   +38.884, E3 +396993.552}
SPL {X  -165.650, Y  +542.772, Z    +0.000, E1   +39.054, E3 +397009.347}
SPL {X  -165.650, Y  +537.647, Z    +0.000, E1   +38.838, E3 +397023.510}
SPL {X  -165.650, Y  +532.636, Z    +0.000, E1   +39.009, E3 +397035.156}
SPL {X  -165.650, Y  +528.320, Z    +0.000, E1   +38.809, E3 +397047.339}
SPL {X  -165.650, Y  +522.377, Z    +0.000, E1   +38.974, E3 +397061.459}
ENDSPLINE

SPLINE
SPL {X  -165.650, Y  +541.168, Z    +0.000, E1   +27.957, E3 +397073.799}
ENDSPLINE

SPLINE
SPL {X  -165.650, Y  +536.052, Z    +0.000, E1   +28.653, E3 +397088.434}
SPL {X  -165.650, Y  +530.452, Z    +0.000, E1   +29.664, E3 +397101.861}
SPL {X  -165.650, Y  +525.298, Z    +0.000, E1   +30.602, E3 +397113.671}
SPL {X  -165.650, Y  +518.290, Z    +0.000, E1   +31.783, E3 +397129.563}
SPL {X  -165.650, Y  +512.706, Z    +0.000, E1   +32.573, E3 +397142.398}
SPL {X  -165.650, Y  +507.785, Z    +0.000, E1   +33.438, E3 +397152.335}
SPL {X  -165.650, Y  +502.877, Z    +0.000, E1   +34.230, E3 +397162.223}
SPL {X  -165.650, Y  +499.289, Z    +0.000, E1   +34.735, E3 +397169.691}
SPL {X  -165.650, Y  +493.800, Z    +0.000, E1   +35.486, E3 +397181.062}
SPL {X  -165.650, Y  +487.198, Z    +0.000, E1   +36.442, E3 +397193.661}
SPL {X  -165.650, Y  +481.130, Z    +0.000, E1   +37.251, E3 +397205.286}
SPL {X  -165.650, Y  +475.455, Z    +0.000, E1   +37.964, E3 +397215.942}
SPL {X  -165.650, Y  +469.901, Z    +0.000, E1   +38.767, E3 +397225.436}
SPL {X  -165.650, Y  +465.276, Z    +0.000, E1   +39.067, E3 +397235.313}
SPL {X  -165.650, Y  +459.623, Z    +0.000, E1   +39.919, E3 +397244.249}
SPL {X  -165.650, Y  +455.681, Z    +0.000, E1   +39.641, E3 +397255.569}
SPL {X  -165.650, Y  +451.332, Z    +0.000, E1   +39.738, E3 +397265.701}
SPL {X  -165.650, Y  +448.050, Z    +0.000, E1   +39.392, E3 +397275.867}
SPL {X  -165.650, Y  +442.946, Z    +0.000, E1   +39.866, E3 +397285.641}
SPL {X  -165.650, Y  +439.091, Z    +0.000, E1   +39.674, E3 +397296.259}
SPL {X  -165.650, Y  +434.131, Z    +0.000, E1   +39.643, E3 +397308.772}
SPL {X  -165.650, Y  +428.810, Z    +0.000, E1   +39.691, E3 +397321.534}
SPL {X  -165.650, Y  +424.197, Z    +0.000, E1   +39.695, E3 +397332.893}
SPL {X  -165.650, Y  +420.220, Z    +0.000, E1   +39.526, E3 +397343.688}
SPL {X  -165.650, Y  +414.177, Z    +0.000, E1   +39.693, E3 +397357.815}
SPL {X  -165.650, Y  +407.394, Z    +0.000, E1   +39.797, E3 +397373.769}
SPL {X  -165.650, Y  +402.798, Z    +0.000, E1   +39.651, E3 +397385.891}
SPL {X  -165.650, Y  +398.253, Z    +0.000, E1   +39.688, E3 +397396.895}
SPL {X  -165.650, Y  +393.720, Z    +0.000, E1   +39.686, E3 +397408.069}
SPL {X  -165.650, Y  +389.210, Z    +0.000, E1   +39.696, E3 +397419.118}
SPL {X  -165.650, Y  +384.878, Z    +0.000, E1   +39.631, E3 +397430.195}
SPL {X  -165.650, Y  +380.529, Z    +0.000, E1   +39.528, E3 +397441.581}
SPL {X  -165.618, Y  +375.240, Z    +0.000, E1   +39.617, E3 +397454.176}
SPL {X  -165.428, Y  +369.922, Z    +0.000, E1   +39.705, E3 +397466.717}
SPL {X  -165.055, Y  +364.469, Z    +0.000, E1   +39.623, E3 +397480.759}
SPL {X  -164.424, Y  +358.387, Z    +0.000, E1   +39.525, E3 +397496.283}
SPL {X  -163.775, Y  +353.645, Z    +0.000, E1   +39.313, E3 +397509.163}
SPL {X  -162.932, Y  +348.615, Z    +0.000, E1   +39.259, E3 +397521.927}
SPL {X  -162.143, Y  +344.596, Z    +0.000, E1   +39.019, E3 +397533.143}
SPL {X  -161.093, Y  +339.912, Z    +0.000, E1   +38.966, E3 +397545.094}
SPL {X  -159.926, Y  +335.332, Z    +0.000, E1   +38.809, E3 +397557.148}
SPL {X  -153.020, Y  +315.059, Z    +0.000, E1   +45.580, E3 +397563.879}
SPL {X  -148.632, Y  +305.368, Z    +0.000, E1   +40.700, E3 +397623.481}
SPL {X  -145.004, Y  +298.414, Z    +0.000, E1   +40.971, E3 +397648.216}
ENDSPLINE

SPLINE
SPL {X  -149.687, Y  +307.551, Z    +0.000, E1   +36.303, E3 +397683.649}
SPL {X  -158.807, Y  +331.381, Z    +0.000, E1   +26.928, E3 +397707.301}
SPL {X  -164.505, Y  +359.058, Z    +0.000, E1   +13.887, E3 +397696.063}
SPL {X  -165.334, Y  +368.271, Z    +0.000, E1    +8.886, E3 +397693.901}
SPL {X  -165.596, Y  +374.277, Z    +0.000, E1    +5.306, E3 +397695.283}
SPL {X  -165.650, Y  +379.419, Z    +0.000, E1    +2.065, E3 +397692.305}
SPL {X  -165.650, Y  +383.176, Z    +0.000, E1    -0.610, E3 +397693.300}
SPL {X  -165.650, Y  +387.435, Z    +0.000, E1    -4.104, E3 +397691.660}
SPL {X  -165.650, Y  +393.422, Z    +0.000, E1    -9.605, E3 +397692.217}
SPL {X  -165.650, Y  +400.450, Z    +0.000, E1   -18.287, E3 +397684.032}
SPL {X  -165.650, Y  +409.248, Z    +0.000, E1   -26.478, E3 +397687.655}
SPL {X  -165.650, Y  +418.660, Z    +0.000, E1   -36.186, E3 +397685.131}
SPL {X  -165.650, Y  +444.260, Z    +0.000, E1   -47.328, E3 +397700.878}
SPL {X  -165.650, Y  +458.981, Z    +0.000, E1   -49.189, E3 +397716.422}
SPL {X  -165.650, Y  +493.049, Z    +0.000, E1   -51.657, E3 +397755.455}
ENDSPLINE

SPLINE
SPL {X  -165.650, Y  +468.984, Z    +0.000, E1   -41.461, E3 +397768.315}
SPL {X  -165.650, Y  +467.052, Z    +0.000, E1   -38.928, E3 +397778.930}
ENDSPLINE

SPLINE
SPL {X  -165.650, Y  +471.956, Z    +0.000, E1   -39.047, E3 +397790.581}
SPL {X  -165.650, Y  +476.270, Z    +0.000, E1   -39.142, E3 +397800.837}
SPL {X  -165.650, Y  +479.585, Z    +0.000, E1   -39.047, E3 +397809.749}
SPL {X  -165.650, Y  +484.115, Z    +0.000, E1   -39.050, E3 +397821.227}
SPL {X  -165.650, Y  +490.374, Z    +0.000, E1   -39.169, E3 +397836.346}
SPL {X  -165.650, Y  +495.141, Z    +0.000, E1   -39.109, E3 +397848.502}
SPL {X  -165.650, Y  +499.941, Z    +0.000, E1   -39.068, E3 +397861.031}
SPL {X  -165.650, Y  +505.989, Z    +0.000, E1   -39.067, E3 +397876.211}
SPL {X  -165.650, Y  +512.188, Z    +0.000, E1   -39.077, E3 +397891.854}
SPL {X  -165.650, Y  +516.634, Z    +0.000, E1   -39.035, E3 +397903.100}
SPL {X  -165.650, Y  +521.541, Z    +0.000, E1   -39.052, E3 +397915.647}
SPL {X  -165.650, Y  +527.474, Z    +0.000, E1   -39.169, E3 +397929.664}
SPL {X  -165.650, Y  +532.836, Z    +0.000, E1   -39.150, E3 +397943.447}
SPL {X  -165.650, Y  +537.667, Z    +0.000, E1   -38.986, E3 +397956.392}
SPL {X  -165.650, Y  +541.183, Z    +0.000, E1   -39.101, E3 +397964.579}
SPL {X  -165.650, Y  +546.018, Z    +0.000, E1   -39.065, E3 +397977.089}
SPL {X  -165.650, Y  +551.666, Z    +0.000, E1   -39.102, E3 +397991.039}
SPL {X  -165.650, Y  +557.612, Z    +0.000, E1   -39.166, E3 +398005.685}
SPL {X  -165.650, Y  +562.850, Z    +0.000, E1   -38.959, E3 +398020.044}
SPL {X  -165.650, Y  +568.257, Z    +0.000, E1   -39.077, E3 +398032.999}
SPL {X  -165.650, Y  +573.200, Z    +0.000, E1   -39.061, E3 +398045.534}
SPL {X  -165.650, Y  +578.240, Z    +0.000, E1   -39.117, E3 +398057.875}
SPL {X  -165.650, Y  +582.804, Z    +0.000, E1   -39.080, E3 +398069.582}
SPL {X  -165.650, Y  +587.640, Z    +0.000, E1   -39.069, E3 +398081.838}
SPL {X  -165.650, Y  +592.685, Z    +0.000, E1   -39.263, E3 +398093.303}
SPL {X  -165.650, Y  +596.539, Z    +0.000, E1   -39.049, E3 +398104.292}
SPL {X  -165.650, Y  +599.973, Z    +0.000, E1   -38.814, E3 +398114.345}
SPL {X  -165.650, Y  +604.635, Z    +0.000, E1   -39.163, E3 +398124.038}
SPL {X  -165.650, Y  +608.365, Z    +0.000, E1   -39.063, E3 +398134.029}
SPL {X  -165.650, Y  +613.618, Z    +0.000, E1   -39.137, E3 +398146.893}
SPL {X  -165.650, Y  +619.584, Z    +0.000, E1   -39.045, E3 +398162.530}
SPL {X  -165.650, Y  +625.662, Z    +0.000, E1   -39.189, E3 +398176.843}
SPL {X  -165.650, Y  +629.982, Z    +0.000, E1   -39.063, E3 +398188.445}
SPL {X  -165.650, Y  +635.019, Z    +0.000, E1   -39.106, E3 +398200.927}
SPL {X  -165.650, Y  +640.403, Z    +0.000, E1   -39.127, E3 +398214.323}
SPL {X  -165.650, Y  +643.707, Z    +0.000, E1   -38.911, E3 +398223.861}
SPL {X  -165.650, Y  +648.294, Z    +0.000, E1   -39.142, E3 +398234.116}
SPL {X  -165.650, Y  +652.477, Z    +0.000, E1   -39.068, E3 +398245.019}
SPL {X  -165.650, Y  +656.920, Z    +0.000, E1   -39.120, E3 +398255.974}
SPL {X  -165.650, Y  +662.945, Z    +0.000, E1   -39.141, E3 +398271.079}
SPL {X  -165.650, Y  +668.296, Z    +0.000, E1   -39.077, E3 +398284.804}
SPL {X  -165.650, Y  +673.138, Z    +0.000, E1   -39.196, E3 +398296.260}
SPL {X  -165.640, Y  +677.281, Z    +0.000, E1   -38.803, E3 +398309.148}
SPL {X  -165.461, Y  +683.414, Z    +0.000, E1   -39.212, E3 +398322.133}
SPL {X  -165.139, Y  +688.497, Z    +0.000, E1   -39.013, E3 +398336.185}
SPL {X  -164.582, Y  +694.282, Z    +0.000, E1   -38.975, E3 +398350.932}
SPL {X  -163.926, Y  +699.336, Z    +0.000, E1   -38.767, E3 +398364.911}
SPL {X  -162.937, Y  +705.358, Z    +0.000, E1   -38.703, E3 +398380.494}
SPL {X  -161.983, Y  +710.160, Z    +0.000, E1   -38.439, E3 +398393.988}
SPL {X  -160.874, Y  +714.989, Z    +0.000, E1   -38.205, E3 +398407.649}
SPL {X  -158.364, Y  +724.087, Z    +0.000, E1   -39.961, E3 +398419.855}
SPL {X  -138.706, Y  +766.057, Z    +0.000, E1   -46.957, E3 +398470.846}
ENDSPLINE

SPLINE
SPL {X  -141.948, Y  +760.885, Z    +0.000, E1   -42.258, E3 +398510.597}
SPL {X  -160.264, Y  +717.397, Z    +0.000, E1   -24.835, E3 +398551.781}
SPL {X  -164.762, Y  +692.628, Z    +0.000, E1   -12.660, E3 +398555.034}
SPL {X  -165.581, Y  +680.274, Z    +0.000, E1    -5.699, E3 +398550.518}
SPL {X  -165.650, Y  +672.825, Z    +0.000, E1    -0.909, E3 +398548.707}
SPL {X  -165.650, Y  +667.803, Z    +0.000, E1    +2.989, E3 +398548.167}
SPL {X  -165.650, Y  +662.773, Z    +0.000, E1    +7.549, E3 +398548.089}
SPL {X  -165.650, Y  +656.581, Z    +0.000, E1   +13.870, E3 +398546.139}
SPL {X  -165.650, Y  +648.120, Z    +0.000, E1   +22.794, E3 +398545.370}
SPL {X  -165.650, Y  +632.103, Z    +0.000, E1   +42.949, E3 +398532.328}
SPL {X  -165.650, Y  +608.448, Z    +0.000, E1   +47.265, E3 +398558.767}
SPL {X  -165.650, Y  +595.526, Z    +0.000, E1   +48.856, E3 +398572.625}
SPL {X  -165.650, Y  +568.828, Z    +0.000, E1   +48.639, E3 +398615.179}
ENDSPLINE

SPLINE
SPL {X  -165.650, Y  +586.972, Z    +0.000, E1   +40.422, E3 +398625.878}
ENDSPLINE

SPLINE
SPL {X  -165.650, Y  +585.370, Z    +0.000, E1   +38.910, E3 +398639.138}
SPL {X  -165.650, Y  +580.805, Z    +0.000, E1   +38.877, E3 +398650.760}
SPL {X  -165.650, Y  +575.679, Z    +0.000, E1   +38.947, E3 +398663.482}
SPL {X  -165.650, Y  +569.616, Z    +0.000, E1   +38.966, E3 +398678.640}
SPL {X  -165.650, Y  +564.364, Z    +0.000, E1   +38.909, E3 +398692.293}
SPL {X  -165.650, Y  +559.065, Z    +0.000, E1   +38.883, E3 +398705.871}
SPL {X  -165.650, Y  +552.770, Z    +0.000, E1   +38.963, E3 +398721.432}
SPL {X  -165.650, Y  +546.277, Z    +0.000, E1   +38.910, E3 +398738.174}
SPL {X  -165.650, Y  +540.151, Z    +0.000, E1   +38.996, E3 +398753.103}
SPL {X  -165.650, Y  +534.008, Z    +0.000, E1   +38.962, E3 +398768.945}
SPL {X  -165.650, Y  +528.320, Z    +0.000, E1   +38.809, E3 +398784.182}
SPL {X  -165.650, Y  +524.195, Z    +0.000, E1   +38.844, E3 +398794.357}
SPL {X  -165.650, Y  +520.666, Z    +0.000, E1   +39.043, E3 +398802.083}
ENDSPLINE

SPLINE
SPL {X  -165.650, Y  +539.854, Z    +0.000, E1   +28.090, E3 +398814.918}
ENDSPLINE

SPLINE
SPL {X  -165.650, Y  +534.443, Z    +0.000, E1   +28.969, E3 +398828.970}
SPL {X  -165.650, Y  +530.452, Z    +0.000, E1   +29.664, E3 +398838.703}
SPL {X  -165.650, Y  +525.298, Z    +0.000, E1   +30.602, E3 +398850.513}
SPL {X  -165.650, Y  +518.290, Z    +0.000, E1   +31.783, E3 +398866.405}
SPL {X  -165.650, Y  +512.706, Z    +0.000, E1   +32.573, E3 +398879.240}
SPL {X  -165.650, Y  +507.785, Z    +0.000, E1   +33.438, E3 +398889.177}
SPL {X  -165.650, Y  +501.257, Z    +0.000, E1   +34.478, E3 +398902.416}
SPL {X  -165.650, Y  +493.800, Z    +0.000, E1   +35.486, E3 +398917.904}
SPL {X  -165.650, Y  +485.583, Z    +0.000, E1   +36.670, E3 +398933.628}
SPL {X  -165.650, Y  +477.375, Z    +0.000, E1   +37.747, E3 +398949.147}
SPL {X  -165.650, Y  +469.901, Z    +0.000, E1   +38.767, E3 +398962.278}
SPL {X  -165.650, Y  +461.805, Z    +0.000, E1   +39.619, E3 +398977.622}
SPL {X  -165.650, Y  +455.681, Z    +0.000, E1   +39.641, E3 +398992.411}
SPL {X  -165.650, Y  +451.332, Z    +0.000, E1   +39.738, E3 +399002.543}
SPL {X  -165.650, Y  +448.050, Z    +0.000, E1   +39.392, E3 +399012.709}
SPL {X  -165.650, Y  +442.946, Z    +0.000, E1   +39.866, E3 +399022.483}
SPL {X  -165.650, Y  +439.091, Z    +0.000, E1   +39.674, E3 +399033.101}
SPL {X  -165.650, Y  +434.131, Z    +0.000, E1   +39.643, E3 +399045.614}
SPL {X  -165.650, Y  +428.810, Z    +0.000, E1   +39.691, E3 +399058.376}
SPL {X  -165.650, Y  +424.197, Z    +0.000, E1   +39.695, E3 +399069.735}
SPL {X  -165.650, Y  +420.220, Z    +0.000, E1   +39.526, E3 +399080.530}
SPL {X  -165.650, Y  +414.177, Z    +0.000, E1   +39.693, E3 +399094.657}
SPL {X  -165.650, Y  +407.394, Z    +0.000, E1   +39.797, E3 +399110.611}
SPL {X  -165.650, Y  +402.798, Z    +0.000, E1   +39.651, E3 +399122.733}
SPL {X  -165.650, Y  +398.253, Z    +0.000, E1   +39.688, E3 +399133.737}
SPL {X  -165.650, Y  +393.720, Z    +0.000, E1   +39.686, E3 +399144.911}
SPL {X  -165.650, Y  +389.210, Z    +0.000, E1   +39.696, E3 +399155.960}
SPL {X  -165.650, Y  +384.878, Z    +0.000, E1   +39.631, E3 +399167.037}
SPL {X  -165.650, Y  +380.529, Z    +0.000, E1   +39.528, E3 +399178.423}
SPL {X  -165.618, Y  +375.240, Z    +0.000, E1   +39.617, E3 +399191.018}
SPL {X  -165.428, Y  +369.922, Z    +0.000, E1   +39.705, E3 +399203.559}
SPL {X  -165.216, Y  +366.519, Z    +0.000, E1   +39.498, E3 +399213.126}
SPL {X  -164.790, Y  +361.646, Z    +0.000, E1   +39.684, E3 +399224.120}
SPL {X  -164.317, Y  +357.530, Z    +0.000, E1   +39.402, E3 +399235.834}
SPL {X  -163.775, Y  +353.645, Z    +0.000, E1   +39.313, E3 +399246.005}
SPL {X  -162.932, Y  +348.615, Z    +0.000, E1   +39.259, E3 +399258.769}
SPL {X  -161.858, Y  +343.258, Z    +0.000, E1   +39.040, E3 +399273.307}
SPL {X  -160.812, Y  +338.758, Z    +0.000, E1   +38.898, E3 +399285.032}
SPL {X  -159.926, Y  +335.332, Z    +0.000, E1   +38.809, E3 +399293.990}
SPL {X  -153.020, Y  +315.059, Z    +0.000, E1   +45.580, E3 +399300.721}
SPL {X  -148.632, Y  +305.368, Z    +0.000, E1   +40.700, E3 +399360.323}
SPL {X  -145.004, Y  +298.414, Z    +0.000, E1   +40.971, E3 +399385.058}
ENDSPLINE

SPLINE
SPL {X  -149.687, Y  +307.551, Z    +0.000, E1   +36.303, E3 +399420.491}
SPL {X  -158.807, Y  +331.381, Z    +0.000, E1   +26.928, E3 +399444.143}
SPL {X  -164.505, Y  +359.058, Z    +0.000, E1   +13.887, E3 +399432.905}
SPL {X  -165.494, Y  +371.321, Z    +0.000, E1    +7.176, E3 +399431.466}
SPL {X  -165.650, Y  +379.419, Z    +0.000, E1    +2.065, E3 +399429.147}
SPL {X  -165.650, Y  +383.176, Z    +0.000, E1    -0.610, E3 +399430.142}
SPL {X  -165.650, Y  +388.696, Z    +0.000, E1    -5.134, E3 +399428.419}
SPL {X  -165.650, Y  +394.663, Z    +0.000, E1   -10.843, E3 +399429.574}
SPL {X  -165.650, Y  +400.450, Z    +0.000, E1   -18.287, E3 +399420.874}
SPL {X  -165.650, Y  +409.248, Z    +0.000, E1   -26.478, E3 +399424.497}
SPL {X  -165.650, Y  +418.660, Z    +0.000, E1   -36.186, E3 +399421.973}
SPL {X  -165.650, Y  +444.260, Z    +0.000, E1   -47.328, E3 +399437.720}
SPL {X  -165.650, Y  +458.981, Z    +0.000, E1   -49.189, E3 +399453.264}
SPL {X  -165.650, Y  +493.049, Z    +0.000, E1   -51.657, E3 +399492.297}
ENDSPLINE

SPLINE
SPL {X  -165.650, Y  +468.984, Z    +0.000, E1   -41.461, E3 +399505.157}
SPL {X  -165.650, Y  +467.052, Z    +0.000, E1   -38.928, E3 +399515.772}
ENDSPLINE

SPLINE
SPL {X  -165.650, Y  +471.956, Z    +0.000, E1   -39.047, E3 +399527.423}
SPL {X  -165.650, Y  +476.270, Z    +0.000, E1   -39.142, E3 +399537.680}
SPL {X  -165.650, Y  +480.876, Z    +0.000, E1   -39.050, E3 +399549.961}
SPL {X  -165.650, Y  +487.054, Z    +0.000, E1   -39.118, E3 +399565.100}
SPL {X  -165.650, Y  +491.785, Z    +0.000, E1   -39.157, E3 +399576.649}
SPL {X  -165.650, Y  +496.519, Z    +0.000, E1   -39.062, E3 +399589.264}
SPL {X  -165.650, Y  +502.351, Z    +0.000, E1   -39.056, E3 +399603.986}
SPL {X  -165.650, Y  +508.180, Z    +0.000, E1   -39.157, E3 +399618.052}
SPL {X  -165.650, Y  +514.341, Z    +0.000, E1   -39.047, E3 +399634.304}
SPL {X  -165.650, Y  +521.541, Z    +0.000, E1   -39.052, E3 +399652.489}
SPL {X  -165.650, Y  +528.401, Z    +0.000, E1   -39.135, E3 +399669.157}
SPL {X  -165.650, Y  +533.857, Z    +0.000, E1   -39.163, E3 +399682.662}
SPL {X  -165.650, Y  +539.651, Z    +0.000, E1   -39.087, E3 +399697.806}
SPL {X  -165.650, Y  +546.018, Z    +0.000, E1   -39.065, E3 +399713.931}
SPL {X  -165.650, Y  +551.666, Z    +0.000, E1   -39.102, E3 +399727.881}
SPL {X  -165.650, Y  +557.612, Z    +0.000, E1   -39.166, E3 +399742.527}
SPL {X  -165.650, Y  +562.850, Z    +0.000, E1   -38.959, E3 +399756.886}
SPL {X  -165.650, Y  +568.257, Z    +0.000, E1   -39.077, E3 +399769.841}
SPL {X  -165.650, Y  +573.200, Z    +0.000, E1   -39.061, E3 +399782.376}
SPL {X  -165.650, Y  +578.240, Z    +0.000, E1   -39.117, E3 +399794.717}
SPL {X  -165.650, Y  +582.804, Z    +0.000, E1   -39.080, E3 +399806.424}
SPL {X  -165.650, Y  +587.640, Z    +0.000, E1   -39.069, E3 +399818.680}
SPL {X  -165.650, Y  +592.685, Z    +0.000, E1   -39.263, E3 +399830.145}
SPL {X  -165.650, Y  +596.539, Z    +0.000, E1   -39.049, E3 +399841.134}
SPL {X  -165.650, Y  +599.973, Z    +0.000, E1   -38.814, E3 +399851.187}
SPL {X  -165.650, Y  +604.635, Z    +0.000, E1   -39.163, E3 +399860.881}
SPL {X  -165.650, Y  +608.365, Z    +0.000, E1   -39.063, E3 +399870.871}
SPL {X  -165.650, Y  +613.618, Z    +0.000, E1   -39.137, E3 +399883.735}
SPL {X  -165.650, Y  +619.584, Z    +0.000, E1   -39.045, E3 +399899.372}
SPL {X  -165.650, Y  +625.662, Z    +0.000, E1   -39.189, E3 +399913.685}
SPL {X  -165.650, Y  +629.982, Z    +0.000, E1   -39.063, E3 +399925.287}
SPL {X  -165.650, Y  +635.019, Z    +0.000, E1   -39.106, E3 +399937.769}
SPL {X  -165.650, Y  +641.706, Z    +0.000, E1   -39.097, E3 +399954.836}
SPL {X  -165.650, Y  +648.294, Z    +0.000, E1   -39.142, E3 +399970.958}
SPL {X  -165.650, Y  +652.477, Z    +0.000, E1   -39.068, E3 +399981.861}
SPL {X  -165.650, Y  +656.920, Z    +0.000, E1   -39.120, E3 +399992.816}
SPL {X  -165.650, Y  +662.945, Z    +0.000, E1   -39.141, E3 +400007.921}
SPL {X  -165.650, Y  +668.296, Z    +0.000, E1   -39.077, E3 +400021.646}
SPL {X  -165.650, Y  +674.193, Z    +0.000, E1   -39.034, E3 +400036.988}
SPL {X  -165.521, Y  +682.029, Z    +0.000, E1   -39.160, E3 +400055.956}
SPL {X  -165.241, Y  +687.126, Z    +0.000, E1   -39.221, E3 +400068.117}
SPL {X  -165.072, Y  +689.330, Z    +0.000, E1   -38.812, E3 +400076.166}
SPL {X  -164.582, Y  +694.282, Z    +0.000, E1   -38.975, E3 +400087.774}
SPL {X  -163.926, Y  +699.336, Z    +0.000, E1   -38.767, E3 +400101.753}
SPL {X  -163.214, Y  +703.806, Z    +0.000, E1   -38.755, E3 +400112.938}
SPL {X  -162.700, Y  +706.623, Z    +0.000, E1   -38.580, E3 +400121.050}
SPL {X  -161.983, Y  +710.160, Z    +0.000, E1   -38.439, E3 +400130.830}
SPL {X  -161.163, Y  +713.794, Z    +0.000, E1   -38.390, E3 +400140.200}
SPL {X  -160.158, Y  +717.801, Z    +0.000, E1   -38.225, E3 +400151.330}
SPL {X  -155.870, Y  +731.575, Z    +0.000, E1   -42.661, E3 +400158.793}
SPL {X  -137.799, Y  +767.431, Z    +0.000, E1   -46.550, E3 +400215.303}
ENDSPLINE

SPLINE
SPL {X  -141.948, Y  +760.885, Z    +0.000, E1   -42.258, E3 +400247.439}
SPL {X  -160.264, Y  +717.397, Z    +0.000, E1   -24.835, E3 +400288.623}
SPL {X  -164.457, Y  +695.345, Z    +0.000, E1   -14.031, E3 +400295.565}
SPL {X  -165.312, Y  +686.072, Z    +0.000, E1    -9.096, E3 +400288.659}
SPL {X  -165.649, Y  +676.021, Z    +0.000, E1    -3.061, E3 +400286.088}
SPL {X  -165.650, Y  +670.589, Z    +0.000, E1    +0.778, E3 +400285.325}
SPL {X  -165.650, Y  +666.842, Z    +0.000, E1    +3.871, E3 +400284.786}
SPL {X  -165.650, Y  +662.773, Z    +0.000, E1    +7.549, E3 +400284.931}
SPL {X  -165.650, Y  +656.581, Z    +0.000, E1   +13.870, E3 +400282.981}
SPL {X  -165.650, Y  +648.120, Z    +0.000, E1   +22.794, E3 +400282.212}
SPL {X  -165.650, Y  +632.103, Z    +0.000, E1   +42.949, E3 +400269.170}
SPL {X  -165.650, Y  +608.448, Z    +0.000, E1   +47.265, E3 +400295.609}
SPL {X  -165.650, Y  +595.526, Z    +0.000, E1   +48.856, E3 +400309.468}
SPL {X  -165.650, Y  +568.828, Z    +0.000, E1   +48.639, E3 +400352.021}
ENDSPLINE

SPLINE
SPL {X  -165.650, Y  +586.972, Z    +0.000, E1   +40.422, E3 +400362.720}
ENDSPLINE

SPLINE
SPL {X  -165.650, Y  +585.370, Z    +0.000, E1   +38.910, E3 +400375.980}
SPL {X  -165.650, Y  +580.805, Z    +0.000, E1   +38.877, E3 +400387.602}
SPL {X  -165.650, Y  +576.923, Z    +0.000, E1   +38.908, E3 +400397.279}
SPL {X  -165.650, Y  +571.957, Z    +0.000, E1   +38.951, E3 +400409.684}
SPL {X  -165.650, Y  +565.217, Z    +0.000, E1   +38.965, E3 +400426.773}
SPL {X  -165.650, Y  +559.065, Z    +0.000, E1   +38.883, E3 +400442.713}
SPL {X  -165.650, Y  +554.358, Z    +0.000, E1   +38.887, E3 +400454.555}
SPL {X  -165.650, Y  +549.409, Z    +0.000, E1   +38.884, E3 +400467.236}
SPL {X  -165.650, Y  +544.480, Z    +0.000, E1   +38.998, E3 +400478.899}
SPL {X  -165.650, Y  +541.194, Z    +0.000, E1   +39.037, E3 +400486.948}
SPL {X  -165.650, Y  +537.647, Z    +0.000, E1   +38.838, E3 +400497.194}
SPL {X  -165.650, Y  +532.636, Z    +0.000, E1   +39.009, E3 +400508.840}
SPL {X  -165.650, Y  +528.320, Z    +0.000, E1   +38.809, E3 +400521.024}
SPL {X  -165.650, Y  +522.377, Z    +0.000, E1   +38.974, E3 +400535.143}
ENDSPLINE

SPLINE
SPL {X  -165.650, Y  +541.168, Z    +0.000, E1   +27.957, E3 +400547.483}
ENDSPLINE

SPLINE
SPL {X  -165.650, Y  +536.052, Z    +0.000, E1   +28.653, E3 +400562.118}
SPL {X  -165.650, Y  +530.452, Z    +0.000, E1   +29.664, E3 +400575.545}
SPL {X  -165.650, Y  +523.712, Z    +0.000, E1   +30.911, E3 +400590.827}
SPL {X  -165.650, Y  +516.975, Z    +0.000, E1   +31.942, E3 +400606.421}
SPL {X  -165.650, Y  +512.706, Z    +0.000, E1   +32.573, E3 +400616.082}
SPL {X  -165.650, Y  +507.785, Z    +0.000, E1   +33.438, E3 +400626.019}
SPL {X  -165.650, Y  +501.257, Z    +0.000, E1   +34.478, E3 +400639.258}
SPL {X  -165.650, Y  +495.236, Z    +0.000, E1   +35.288, E3 +400651.764}
SPL {X  -165.650, Y  +488.684, Z    +0.000, E1   +36.217, E3 +400664.661}
SPL {X  -165.650, Y  +481.130, Z    +0.000, E1   +37.251, E3 +400678.970}
SPL {X  -165.650, Y  +475.455, Z    +0.000, E1   +37.964, E3 +400689.626}
SPL {X  -165.650, Y  +469.901, Z    +0.000, E1   +38.767, E3 +400699.121}
SPL {X  -165.650, Y  +465.276, Z    +0.000, E1   +39.067, E3 +400708.997}
SPL {X  -165.650, Y  +459.623, Z    +0.000, E1   +39.919, E3 +400717.933}
SPL {X  -165.650, Y  +455.681, Z    +0.000, E1   +39.641, E3 +400729.253}
SPL {X  -165.650, Y  +451.332, Z    +0.000, E1   +39.738, E3 +400739.385}
SPL {X  -165.650, Y  +448.050, Z    +0.000, E1   +39.392, E3 +400749.551}
SPL {X  -165.650, Y  +442.946, Z    +0.000, E1   +39.866, E3 +400759.326}
SPL {X  -165.650, Y  +439.091, Z    +0.000, E1   +39.674, E3 +400769.944}
SPL {X  -165.650, Y  +435.404, Z    +0.000, E1   +39.549, E3 +400779.781}
SPL {X  -165.650, Y  +429.757, Z    +0.000, E1   +39.737, E3 +400792.730}
SPL {X  -165.650, Y  +424.197, Z    +0.000, E1   +39.695, E3 +400806.577}
SPL {X  -165.650, Y  +420.220, Z    +0.000, E1   +39.526, E3 +400817.372}
SPL {X  -165.650, Y  +415.675, Z    +0.000, E1   +39.706, E3 +400827.534}
SPL {X  -165.650, Y  +412.313, Z    +0.000, E1   +39.567, E3 +400836.611}
SPL {X  -165.650, Y  +407.394, Z    +0.000, E1   +39.797, E3 +400847.454}
SPL {X  -165.650, Y  +402.798, Z    +0.000, E1   +39.651, E3 +400859.575}
SPL {X  -165.650, Y  +398.253, Z    +0.000, E1   +39.688, E3 +400870.579}
SPL {X  -165.650, Y  +393.720, Z    +0.000, E1   +39.686, E3 +400881.753}
SPL {X  -165.650, Y  +389.210, Z    +0.000, E1   +39.696, E3 +400892.803}
SPL {X  -165.650, Y  +384.878, Z    +0.000, E1   +39.631, E3 +400903.879}
SPL {X  -165.650, Y  +378.931, Z    +0.000, E1   +39.598, E3 +400918.976}
SPL {X  -165.490, Y  +371.216, Z    +0.000, E1   +39.708, E3 +400937.348}
SPL {X  -165.055, Y  +364.469, Z    +0.000, E1   +39.623, E3 +400954.443}
SPL {X  -164.424, Y  +358.387, Z    +0.000, E1   +39.525, E3 +400969.967}
SPL {X  -163.775, Y  +353.645, Z    +0.000, E1   +39.313, E3 +400982.847}
SPL {X  -162.932, Y  +348.615, Z    +0.000, E1   +39.259, E3 +400995.611}
SPL {X  -162.143, Y  +344.596, Z    +0.000, E1   +39.019, E3 +401006.828}
SPL {X  -161.093, Y  +339.912, Z    +0.000, E1   +38.966, E3 +401018.778}
SPL {X  -159.926, Y  +335.332, Z    +0.000, E1   +38.809, E3 +401030.832}
SPL {X  -154.584, Y  +318.971, Z    +0.000, E1   +44.936, E3 +401033.463}
SPL {X  -151.650, Y  +311.851, Z    +0.000, E1   +46.071, E3 +401040.998}
SPL {X  -148.632, Y  +305.368, Z    +0.000, E1   +40.700, E3 +401097.165}
SPL {X  -145.004, Y  +298.414, Z    +0.000, E1   +40.971, E3 +401121.900}
ENDSPLINE

SPLINE
SPL {X  -149.687, Y  +307.551, Z    +0.000, E1   +36.303, E3 +401157.333}
SPL {X  -158.807, Y  +331.381, Z    +0.000, E1   +26.928, E3 +401180.985}
SPL {X  -164.505, Y  +359.058, Z    +0.000, E1   +13.887, E3 +401169.747}
SPL {X  -165.494, Y  +371.321, Z    +0.000, E1    +7.176, E3 +401168.308}
SPL {X  -165.650, Y  +379.419, Z    +0.000, E1    +2.065, E3 +401165.989}
SPL {X  -165.650, Y  +383.176, Z    +0.000, E1    -0.610, E3 +401166.984}
SPL {X  -165.650, Y  +388.696, Z    +0.000, E1    -5.134, E3 +401165.261}
SPL {X  -165.650, Y  +394.663, Z    +0.000, E1   -10.843, E3 +401166.416}
SPL {X  -165.650, Y  +400.450, Z    +0.000, E1   -18.287, E3 +401157.716}
SPL {X  -165.650, Y  +409.248, Z    +0.000, E1   -26.478, E3 +401161.339}
SPL {X  -165.650, Y  +418.660, Z    +0.000, E1   -36.186, E3 +401158.815}
SPL {X  -165.650, Y  +444.260, Z    +0.000, E1   -47.328, E3 +401174.563}
SPL {X  -165.650, Y  +458.981, Z    +0.000, E1   -49.189, E3 +401190.106}
SPL {X  -165.650, Y  +493.049, Z    +0.000, E1   -51.657, E3 +401229.139}
ENDSPLINE

SPLINE
SPL {X  -165.650, Y  +468.984, Z    +0.000, E1   -41.461, E3 +401241.999}
SPL {X  -165.650, Y  +467.052, Z    +0.000, E1   -38.928, E3 +401252.614}
ENDSPLINE

SPLINE
SPL {X  -165.650, Y  +471.956, Z    +0.000, E1   -39.047, E3 +401264.265}
SPL {X  -165.650, Y  +476.270, Z    +0.000, E1   -39.142, E3 +401274.522}
SPL {X  -165.650, Y  +480.876, Z    +0.000, E1   -39.050, E3 +401286.804}
SPL {X  -165.650, Y  +487.054, Z    +0.000, E1   -39.118, E3 +401301.943}
SPL {X  -165.650, Y  +491.785, Z    +0.000, E1   -39.157, E3 +401313.492}
SPL {X  -165.650, Y  +496.519, Z    +0.000, E1   -39.062, E3 +401326.106}
SPL {X  -165.650, Y  +502.351, Z    +0.000, E1   -39.056, E3 +401340.828}
SPL {X  -165.650, Y  +508.180, Z    +0.000, E1   -39.157, E3 +401354.895}
SPL {X  -165.650, Y  +513.074, Z    +0.000, E1   -38.997, E3 +401368.112}
SPL {X  -165.650, Y  +518.439, Z    +0.000, E1   -39.071, E3 +401381.263}
SPL {X  -165.650, Y  +523.032, Z    +0.000, E1   -38.966, E3 +401393.399}
SPL {X  -165.650, Y  +528.401, Z    +0.000, E1   -39.135, E3 +401405.999}
SPL {X  -165.650, Y  +533.857, Z    +0.000, E1   -39.163, E3 +401419.505}
SPL {X  -165.650, Y  +539.651, Z    +0.000, E1   -39.087, E3 +401434.649}
SPL {X  -165.650, Y  +544.603, Z    +0.000, E1   -39.103, E3 +401446.824}
SPL {X  -165.650, Y  +547.280, Z    +0.000, E1   -38.965, E3 +401454.404}
SPL {X  -165.650, Y  +551.666, Z    +0.000, E1   -39.102, E3 +401464.723}
SPL {X  -165.650, Y  +555.880, Z    +0.000, E1   -39.094, E3 +401475.294}
SPL {X  -165.650, Y  +559.255, Z    +0.000, E1   -39.167, E3 +401483.330}
SPL {X  -165.650, Y  +562.850, Z    +0.000, E1   -38.959, E3 +401493.728}
SPL {X  -165.650, Y  +568.257, Z    +0.000, E1   -39.077, E3 +401506.683}
SPL {X  -165.650, Y  +573.200, Z    +0.000, E1   -39.061, E3 +401519.218}
SPL {X  -165.650, Y  +578.240, Z    +0.000, E1   -39.117, E3 +401531.559}
SPL {X  -165.650, Y  +582.804, Z    +0.000, E1   -39.080, E3 +401543.266}
SPL {X  -165.650, Y  +587.640, Z    +0.000, E1   -39.069, E3 +401555.523}
SPL {X  -165.650, Y  +592.685, Z    +0.000, E1   -39.263, E3 +401566.987}
SPL {X  -165.650, Y  +596.539, Z    +0.000, E1   -39.049, E3 +401577.976}
SPL {X  -165.650, Y  +599.973, Z    +0.000, E1   -38.814, E3 +401588.029}
SPL {X  -165.650, Y  +604.635, Z    +0.000, E1   -39.163, E3 +401597.723}
SPL {X  -165.650, Y  +608.365, Z    +0.000, E1   -39.063, E3 +401607.713}
SPL {X  -165.650, Y  +612.142, Z    +0.000, E1   -39.023, E3 +401617.443}
SPL {X  -165.650, Y  +616.635, Z    +0.000, E1   -39.260, E3 +401627.330}
SPL {X  -165.650, Y  +620.299, Z    +0.000, E1   -38.904, E3 +401638.717}
SPL {X  -165.650, Y  +625.662, Z    +0.000, E1   -39.189, E3 +401650.528}
SPL {X  -165.650, Y  +629.982, Z    +0.000, E1   -39.063, E3 +401662.129}
SPL {X  -165.650, Y  +634.317, Z    +0.000, E1   -39.239, E3 +401671.919}
SPL {X  -165.650, Y  +639.215, Z    +0.000, E1   -39.074, E3 +401685.445}
SPL {X  -165.650, Y  +643.707, Z    +0.000, E1   -38.911, E3 +401697.545}
SPL {X  -165.650, Y  +648.294, Z    +0.000, E1   -39.142, E3 +401707.800}
SPL {X  -165.650, Y  +652.477, Z    +0.000, E1   -39.068, E3 +401718.703}
SPL {X  -165.650, Y  +656.920, Z    +0.000, E1   -39.120, E3 +401729.658}
SPL {X  -165.650, Y  +662.945, Z    +0.000, E1   -39.141, E3 +401744.763}
SPL {X  -165.650, Y  +668.296, Z    +0.000, E1   -39.077, E3 +401758.488}
SPL {X  -165.650, Y  +673.138, Z    +0.000, E1   -39.196, E3 +401769.944}
SPL {X  -165.640, Y  +677.281, Z    +0.000, E1   -38.803, E3 +401782.833}
SPL {X  -165.461, Y  +683.414, Z    +0.000, E1   -39.212, E3 +401795.817}
SPL {X  -165.139, Y  +688.497, Z    +0.000, E1   -39.013, E3 +401809.869}
SPL {X  -164.471, Y  +695.227, Z    +0.000, E1   -38.971, E3 +401827.164}
SPL {X  -163.795, Y  +700.218, Z    +0.000, E1   -38.698, E3 +401841.110}
SPL {X  -162.937, Y  +705.358, Z    +0.000, E1   -38.703, E3 +401854.178}
SPL {X  -161.983, Y  +710.160, Z    +0.000, E1   -38.439, E3 +401867.672}
SPL {X  -160.874, Y  +714.989, Z    +0.000, E1   -38.205, E3 +401881.333}
SPL {X  -158.364, Y  +724.087, Z    +0.000, E1   -39.961, E3 +401893.539}
SPL {X  -138.706, Y  +766.057, Z    +0.000, E1   -46.957, E3 +401944.531}
ENDSPLINE

